METHOD PRIVATE DisposeSelfCreatedNodes : BOOL
VAR
	node : I_Node;
END_VAR
WHILE selfCreatedNodes.TryPop(node) DO
	node.Dispose();
END_WHILE
END_METHOD

METHOD PRIVATE RegisterWithDatatypes
VAR_INPUT
END_VAR
IF datatypes = 0 THEN
	RETURN;
END_IF

datatypes.OnEvent('OnDatatypeAdded', THIS^);
END_METHOD

METHOD PROTECTED CreateAliasArrayBundleNode : I_Node
VAR_INPUT
	NodeDatatype : I_AliasDatatype;
END_VAR
VAR
	pAnyBundleNode : POINTER TO AnyAliasArrayBundleNode;
END_VAR
pAnyBundleNode := __NEW(AnyAliasArrayBundleNode(AliasDatatype := NodeDatatype));
CreateAliasArrayBundleNode := pAnyBundleNode^;
END_METHOD

METHOD PROTECTED CreateAliasArrayUnbundleNode : I_Node
VAR_INPUT
	NodeDatatype : I_AliasDatatype;
END_VAR
VAR
	pAnyUnbundleNode : POINTER TO AnyAliasArrayUnbundleNode;
END_VAR
pAnyUnbundleNode := __NEW(AnyAliasArrayUnbundleNode(AliasDatatype := NodeDatatype));
CreateAliasArrayUnbundleNode := pAnyUnbundleNode^;
END_METHOD

METHOD PROTECTED CreateAliasStructureBundleNode : I_Node
VAR_INPUT
	NodeDatatype : I_AliasDatatype;
END_VAR
VAR
	pAnyBundleNode : POINTER TO AnyAliasStructureBundleNode;
END_VAR
pAnyBundleNode := __NEW(AnyAliasStructureBundleNode(AliasDatatype := NodeDatatype));
CreateAliasStructureBundleNode := pAnyBundleNode^;
END_METHOD

METHOD PROTECTED CreateAliasStructureUnbundleNode : I_Node
VAR_INPUT
	NodeDatatype : I_AliasDatatype;
END_VAR
VAR
	pAnyUnbundleNode : POINTER TO AnyAliasStructureUnbundleNode;
END_VAR
pAnyUnbundleNode := __NEW(AnyAliasStructureUnbundleNode(AliasDatatype := NodeDatatype));
CreateAliasStructureUnbundleNode := pAnyUnbundleNode^;
END_METHOD

METHOD PROTECTED CreateArrayBundleNode : I_Node
VAR_INPUT
	NodeDatatype : I_ArrayDatatype;
END_VAR
VAR
	pAnyBundleNode : POINTER TO AnyArrayBundleNode;
END_VAR
pAnyBundleNode := __NEW(AnyArrayBundleNode(ArrayDatatype := NodeDatatype));
CreateArrayBundleNode := pAnyBundleNode^;
END_METHOD

METHOD PROTECTED CreateArrayUnbundleNode : I_Node
VAR_INPUT
	NodeDatatype : I_ArrayDatatype;
END_VAR
VAR
	pAnyUnbundleNode : POINTER TO AnyArrayUnbundleNode;
END_VAR
pAnyUnbundleNode := __NEW(AnyArrayUnbundleNode(ArrayDatatype := NodeDatatype));
CreateArrayUnbundleNode := pAnyUnbundleNode^;
END_METHOD

METHOD PROTECTED CreateDisplayNode : I_Node
VAR_INPUT
	NodeDatatype : I_Datatype;
END_VAR
VAR
	pAnyDisplayNode : POINTER TO AnyDisplayNode;
END_VAR
pAnyDisplayNode := __NEW(AnyDisplayNode(Datatype := NodeDatatype));
CreateDisplayNode := pAnyDisplayNode^;
END_METHOD

METHOD PROTECTED CreateInterfaceDisplayNode : I_Node
VAR_INPUT
	NodeDatatype : I_InterfaceDatatype;
END_VAR
VAR
	pAnyInterfaceDisplayNode : POINTER TO AnyInterfaceDisplayNode;
END_VAR
pAnyInterfaceDisplayNode := __NEW(AnyInterfaceDisplayNode(Datatype := NodeDatatype));
CreateInterfaceDisplayNode := pAnyInterfaceDisplayNode^;
END_METHOD

METHOD PROTECTED CreateLiteralNode : I_Node
VAR_INPUT
	NodeDatatype : I_Datatype;
END_VAR
VAR
	pAnyLiteralNode : POINTER TO AnyLiteralNode;
END_VAR
pAnyLiteralNode := __NEW(AnyLiteralNode(Datatype := NodeDatatype));
CreateLiteralNode := pAnyLiteralNode^;
END_METHOD

METHOD PROTECTED CreateStructureBundleNode : I_Node
VAR_INPUT
	NodeDatatype : I_StructuredDatatype;
END_VAR
VAR
	pAnyBundleNode : POINTER TO AnyStructureBundleNode;
END_VAR
pAnyBundleNode := __NEW(AnyStructureBundleNode(StructuredDatatype := NodeDatatype));
CreateStructureBundleNode := pAnyBundleNode^;
END_METHOD

METHOD PROTECTED CreateStructureUnbundleNode : I_Node
VAR_INPUT
	NodeDatatype : I_StructuredDatatype;
END_VAR
VAR
	pAnyUnbundleNode : POINTER TO AnyStructureUnbundleNode;
END_VAR
pAnyUnbundleNode := __NEW(AnyStructureUnbundleNode(StructuredDatatype := NodeDatatype));
CreateStructureUnbundleNode := pAnyUnbundleNode^;
END_METHOD

METHOD PROTECTED RegisterAliasArrayBundleNodeOfType
VAR_INPUT
	AliasDatatype : I_AliasDatatype;
END_VAR
VAR
	node : I_Node;
	path : T_MAXSTRING;
END_VAR
node := CreateAliasArrayBundleNode(AliasDatatype);
selfCreatedNodes.Push(node);
path := concat('Bundle/', AliasDatatype.Identifier);
nodeFactory.AddNodeAsPrototype(path,node);
END_METHOD

METHOD PROTECTED RegisterAliasArrayUnbundleNodeOfType
VAR_INPUT
	AliasDatatype : I_AliasDatatype;
END_VAR
VAR
	node : I_Node;
	path : T_MAXSTRING;
END_VAR
node := CreateAliasArrayUnbundleNode(AliasDatatype);
selfCreatedNodes.Push(node);
path := concat('Unbundle/', AliasDatatype.Identifier);
nodeFactory.AddNodeAsPrototype(path,node);
END_METHOD

METHOD PROTECTED RegisterAliasStructureBundleNodeOfType
VAR_INPUT
	AliasDatatype : I_AliasDatatype;
END_VAR
VAR
	node : I_Node;
	path : T_MAXSTRING;
END_VAR
node := CreateAliasStructureBundleNode(AliasDatatype);
selfCreatedNodes.Push(node);
path := concat('Bundle/', AliasDatatype.Identifier);
nodeFactory.AddNodeAsPrototype(path,node);
END_METHOD

METHOD PROTECTED RegisterAliasStructureUnbundleNodeOfType
VAR_INPUT
	AliasDatatype : I_AliasDatatype;
END_VAR
VAR
	node : I_Node;
	path : T_MAXSTRING;
END_VAR
node := CreateAliasStructureUnbundleNode(AliasDatatype);
selfCreatedNodes.Push(node);
path := concat('Unbundle/', AliasDatatype.Identifier);
nodeFactory.AddNodeAsPrototype(path,node);
END_METHOD

METHOD PROTECTED RegisterArrayBundleNodeOfType
VAR_INPUT
	NodeDatatype : I_ArrayDatatype;
END_VAR
VAR
	node : I_Node;
	path : T_MAXSTRING;
END_VAR
node := CreateArrayBundleNode(NodeDatatype);
selfCreatedNodes.Push(node);
path := concat('Bundle/', NodeDatatype.Identifier);
nodeFactory.AddNodeAsPrototype(path,node);
END_METHOD

METHOD PROTECTED RegisterArrayUnbundleNodeOfType
VAR_INPUT
	NodeDatatype : I_ArrayDatatype;
END_VAR
VAR
	node : I_Node;
	path : T_MAXSTRING;
END_VAR
node := CreateArrayUnbundleNode(NodeDatatype);
selfCreatedNodes.Push(node);
path := concat('Unbundle/', NodeDatatype.Identifier);
nodeFactory.AddNodeAsPrototype(path,node);
END_METHOD

METHOD PROTECTED RegisterInterfaceDisplayNodeOfType
VAR_INPUT
	NodeDatatype : I_InterfaceDatatype;
END_VAR
VAR
	node : I_Node;
	path : T_MAXSTRING;
END_VAR
node := CreateInterfaceDisplayNode(NodeDatatype);
selfCreatedNodes.Push(node);
path := concat('Display/', NodeDatatype.Identifier);
nodeFactory.AddNodeAsPrototype(path,node);
END_METHOD

METHOD PROTECTED RegisterInterfaceLiteralNodeOfType
VAR_INPUT
	NodeDatatype : I_InterfaceDatatype;
END_VAR
VAR
	node : I_Node;
	path : T_MAXSTRING;
END_VAR
node := CreateLiteralNode(NodeDatatype);
selfCreatedNodes.Push(node);
path := concat('Literal/', NodeDatatype.Identifier);
nodeFactory.AddNodeAsPrototype(path,node);
END_METHOD

METHOD PROTECTED RegisterPrimitiveDisplayNodeOfType
VAR_INPUT
	NodeDatatype : I_Datatype;
END_VAR
VAR
	node : I_Node;
	path : T_MAXSTRING;
END_VAR
node := CreateDisplayNode(NodeDatatype);
selfCreatedNodes.Push(node);
path := concat('Display/', NodeDatatype.TypeName);
nodeFactory.AddNodeAsPrototype(path,node);
END_METHOD

METHOD PROTECTED RegisterPrimitiveLiteralNodeOfType
VAR_INPUT
	NodeDatatype : I_Datatype;
END_VAR
VAR
	node : I_Node;
	path : T_MAXSTRING;
END_VAR
node := CreateLiteralNode(NodeDatatype);
selfCreatedNodes.Push(node);
path := concat('Literal/', NodeDatatype.TypeName);
nodeFactory.AddNodeAsPrototype(path,node);
END_METHOD

METHOD PROTECTED RegisterStructureBundleNodeOfType
VAR_INPUT
	NodeDatatype : I_StructuredDatatype;
END_VAR
VAR
	node : I_Node;
	path : T_MAXSTRING;
END_VAR
node := CreateStructureBundleNode(NodeDatatype);
selfCreatedNodes.Push(node);
path := concat('Bundle/', NodeDatatype.Identifier);
nodeFactory.AddNodeAsPrototype(path,node);
END_METHOD

METHOD PROTECTED RegisterStructureUnbundleNodeOfType
VAR_INPUT
	NodeDatatype : I_StructuredDatatype;
END_VAR
VAR
	node : I_Node;
	path : T_MAXSTRING;
END_VAR
node := CreateStructureUnbundleNode(NodeDatatype);
selfCreatedNodes.Push(node);
path := concat('Unbundle/', NodeDatatype.Identifier);
nodeFactory.AddNodeAsPrototype(path,node);
END_METHOD

METHOD PROTECTED RegisterUdtDisplayNodeOfType
VAR_INPUT
	NodeDatatype : I_UserDefinedDatatype;
END_VAR
VAR
	node : I_Node;
	path : T_MAXSTRING;
END_VAR
node := CreateDisplayNode(NodeDatatype);
selfCreatedNodes.Push(node);
path := concat('Display/', NodeDatatype.Identifier);
nodeFactory.AddNodeAsPrototype(path,node);
END_METHOD

METHOD PROTECTED RegisterUdtLiteralNodeOfType
VAR_INPUT
	NodeDatatype : I_UserDefinedDatatype;
END_VAR
VAR
	node : I_Node;
	path : T_MAXSTRING;
END_VAR
node := CreateLiteralNode(NodeDatatype);
selfCreatedNodes.Push(node);
path := concat('Literal/', NodeDatatype.Identifier);
nodeFactory.AddNodeAsPrototype(path,node);
END_METHOD

METHOD PUBLIC HandleEvent
VAR_INPUT
	Event : I_Event;
END_VAR
VAR
	datatypeAddedEvent : I_DatatypeAddedEvent;
	primitiveDatatype : I_Datatype;
	aliasDatatypeAddedEvent : I_AliasDatatypeAddedEvent;
	aliasDatatype : I_AliasDatatype;
	enumDatatypeAddedEvent : I_EnumDatatypeAddedEvent;
	enumDatatype : I_EnumDatatype;
	structuredDatatypeAddedEvent : I_StructuredDatatypeAddedEvent;
	structureDatatype : I_StructuredDatatype;
	interfaceDatatypeAddedEvent : I_InterfaceDatatypeAddedEvent;
	interfaceDatatype : I_InterfaceDatatype;
	arrayDatatypeAddedEvent : I_ArrayDatatypeAddedEvent;
	arrayDatatype : I_ArrayDatatype;
END_VAR
IF __QUERYINTERFACE(event, aliasDatatypeAddedEvent) THEN
	aliasDatatype := aliasDatatypeAddedEvent.Target;
	RegisterUdtLiteralNodeOfType(aliasDatatype);
	RegisterUdtDisplayNodeOfType(aliasDatatype);
	
	// at this point we have the lowest level alias who's base type is not alias (or we reached a breakout)
	IF aliasDatatype.Root.TryResolveAsArrayDatatype(arrayDatatype) THEN
		RegisterAliasArrayBundleNodeOfType(aliasDatatype);
		RegisterAliasArrayUnbundleNodeOfType(aliasDatatype);
	ELSIF aliasDatatype.Root.TryResolveAsStructuredDatatype(structureDatatype) THEN
		RegisterAliasStructureBundleNodeOfType(aliasDatatype);
		RegisterAliasStructureUnbundleNodeOfType(aliasDatatype);
	END_IF
		
	RETURN;
END_IF

IF __QUERYINTERFACE(event, enumDatatypeAddedEvent) THEN
	enumDatatype := enumDatatypeAddedEvent.Target;
	RegisterUdtLiteralNodeOfType(enumDatatype);
	RegisterUdtDisplayNodeOfType(enumDatatype);
	RETURN;
END_IF

IF __QUERYINTERFACE(event, interfaceDatatypeAddedEvent) THEN
	interfaceDatatype := interfaceDatatypeAddedEvent.Target;
	RegisterInterfaceLiteralNodeOfType(interfaceDatatype);
	RegisterInterfaceDisplayNodeOfType(interfaceDatatype);
	RETURN;
END_IF

IF __QUERYINTERFACE(event, structuredDatatypeAddedEvent) THEN
	structureDatatype := structuredDatatypeAddedEvent.Target;
	RegisterUdtLiteralNodeOfType(structureDatatype);
	RegisterUdtDisplayNodeOfType(structureDatatype);
	RegisterStructureBundleNodeOfType(structureDatatype);
	RegisterStructureUnbundleNodeOfType(structureDatatype);
	RETURN;
END_IF

IF __QUERYINTERFACE(event, arrayDatatypeAddedEvent) THEN
	RegisterUdtLiteralNodeOfType(arrayDatatypeAddedEvent.Target);
	RegisterUdtDisplayNodeOfType(arrayDatatypeAddedEvent.Target);
	RegisterArrayBundleNodeOfType(arrayDatatypeAddedEvent.Target);
	RegisterArrayUnbundleNodeOfType(arrayDatatypeAddedEvent.Target);
	RETURN;
END_IF

IF __QUERYINTERFACE(event, datatypeAddedEvent) THEN
	primitiveDatatype := datatypeAddedEvent.Target;
	RegisterPrimitiveLiteralNodeOfType(primitiveDatatype);
	RegisterPrimitiveDisplayNodeOfType(primitiveDatatype);
	RETURN;
END_IF
END_METHOD

END_FUNCTION_BLOCK

// Node/Bundle/AnyAliasArrayBundleNode
{attribute 'linkalways'} 
{attribute 'no_explicit_call' := 'This FB is a CLASS and must be accessed using methods or properties'}
{attribute 'enable_dynamic_creation'}
FUNCTION_BLOCK FINAL AnyAliasArrayBundleNode EXTENDS Node
VAR
	in : I_AliasDatatype;
	out : I_AliasDatatype;
	datatypeOperations : DatatypeOperations;
	selfMadeElements : Stack;
END_VAR

METHOD FB_init : BOOL
VAR_INPUT
	bInitRetains : BOOL; // if TRUE, the retain variables are initialized (warm start / cold start)
	bInCopyCode : BOOL;  // if TRUE, the instance afterwards gets moved into the copy code (online change)
	AliasDatatype : I_AliasDatatype;
END_VAR
VAR
	inAsArray : I_ArrayDatatype;
	inAs1D : I_ArrayDatatype_1D;
	inAs2D : I_ArrayDatatype_2D;
	inAs3D : I_ArrayDatatype_3D;
END_VAR
AliasDatatype.Clone().TryResolveAsAliasDatatype(out);
AddOutput('out', out);

AliasDatatype.Clone().TryResolveAsAliasDatatype(in);
in.Root.TryResolveAsArrayDatatype(inAsArray);

IF inAsArray.TryResolveAs1DArrayDatatype(inAs1D) THEN
	ConfigureFor1DArray(inAs1D);
ELSIF inAsArray.TryResolveAs2DArrayDatatype(inAs2D) THEN
	ConfigureFor2DArray(inAs2D);
ELSIF inAsArray.TryResolveAs3DArrayDatatype(inAs3D) THEN
	ConfigureFor3DArray(inAs3D);
END_IF
END_METHOD

METHOD FB_exit : BOOL
VAR_INPUT
	bInCopyCode : BOOL; // if TRUE, the exit method is called for exiting an instance that is copied afterwards (online change).
END_VAR
VAR
	element : I_Datatype;
END_VAR
IF bInCopyCode THEN
	RETURN;
END_IF

in.Dispose();
out.Dispose();
datatypeOperations.Clear();

WHILE selfMadeElements.TryPop(element) DO
	IF element <> 0 THEN 
		element.Dispose();
	END_IF
END_WHILE
END_METHOD

METHOD PRIVATE ConfigureFor1DArray
VAR_INPUT
	array1D : I_ArrayDatatype_1D;
END_VAR
VAR
	lowerBound : DINT;
	upperBound : DINT;
	i : DINT;
	element : I_Datatype;
	elementClone : I_Datatype;
END_VAR
IF NOT array1D.TryGetLowerBound(1, lowerBound) THEN
	RETURN;
END_IF

IF NOT array1D.TryGetUpperBound(1, upperBound) THEN
	RETURN;
END_IF

FOR i := lowerBound TO upperBound DO
	
	IF array1D.TryGetElementAsDatatypeByIndex(i, element) THEN
		elementClone := element.Clone();
		datatypeOperations.AddMemoryCopyOperation(elementClone, element);
		AddParameter(Get1DIndexName(i), elementClone);
		selfMadeElements.Push(elementClone);
	END_IF
	
END_FOR
END_METHOD

METHOD PRIVATE ConfigureFor2DArray
VAR_INPUT
	array2D : I_ArrayDatatype_2D;
END_VAR
VAR
	lowerBoundD1 : DINT;
	upperBoundD1 : DINT;
	lowerBoundD2 : DINT;
	upperBoundD2 : DINT;
	i, j : DINT;
	element : I_Datatype;
	elementClone : I_Datatype;
END_VAR
IF NOT array2D.TryGetLowerBound(1, lowerBoundD1) THEN
	RETURN;
END_IF

IF NOT array2D.TryGetUpperBound(1, upperBoundD1) THEN
	RETURN;
END_IF

IF NOT array2D.TryGetLowerBound(2, lowerBoundD2) THEN
	RETURN;
END_IF

IF NOT array2D.TryGetUpperBound(2, upperBoundD2) THEN
	RETURN;
END_IF

FOR i := lowerBoundD1 TO upperBoundD1 DO
	FOR j := lowerBoundD2 TO upperBoundD2 DO
	
		IF array2D.TryGetElementAsDatatypeByIndex(i, j, element) THEN
			elementClone := element.Clone();
			datatypeOperations.AddMemoryCopyOperation(elementClone, element);
			AddParameter(Get2DIndexName(i,j), elementClone);
			selfMadeElements.Push(elementClone);
		END_IF
	
	END_FOR
END_FOR
END_METHOD

METHOD PRIVATE ConfigureFor3DArray
VAR_INPUT
	array3D : I_ArrayDatatype_3D;
END_VAR
VAR
	lowerBoundD1 : DINT;
	upperBoundD1 : DINT;
	lowerBoundD2 : DINT;
	upperBoundD2 : DINT;
	lowerBoundD3 : DINT;
	upperBoundD3 : DINT;
	i, j, k : DINT;
	element : I_Datatype;
	elementClone : I_Datatype;
END_VAR
IF NOT array3D.TryGetLowerBound(1, lowerBoundD1) THEN
	RETURN;
END_IF

IF NOT array3D.TryGetUpperBound(1, upperBoundD1) THEN
	RETURN;
END_IF

IF NOT array3D.TryGetLowerBound(2, lowerBoundD2) THEN
	RETURN;
END_IF

IF NOT array3D.TryGetUpperBound(2, upperBoundD2) THEN
	RETURN;
END_IF

IF NOT array3D.TryGetLowerBound(3, lowerBoundD3) THEN
	RETURN;
END_IF

IF NOT array3D.TryGetUpperBound(3, upperBoundD3) THEN
	RETURN;
END_IF

FOR i := lowerBoundD1 TO upperBoundD1 DO
	FOR j := lowerBoundD2 TO upperBoundD2 DO
		FOR k := lowerBoundD3 TO upperBoundD3 DO
	
			IF array3D.TryGetElementAsDatatypeByIndex(i, j, k, element) THEN
				elementClone := element.Clone();
				datatypeOperations.AddMemoryCopyOperation(elementClone, element);
				AddParameter(Get3DIndexName(i, j, k), elementClone);
				selfMadeElements.Push(elementClone);
			END_IF
			
		END_FOR
	END_FOR
END_FOR
END_METHOD

METHOD PRIVATE Get1DIndexName : T_MAXSTRING
VAR_INPUT
	Index : DINT;
END_VAR
Get1DIndexName := concat('[', DINT_TO_STRING(Index));
Get1DIndexName := concat(Get1DIndexName, ']');
END_METHOD

METHOD PRIVATE Get2DIndexName : T_MAXSTRING
VAR_INPUT
	Index1 : DINT;
	Index2 : DINT;
END_VAR
Get2DIndexName := concat('[', DINT_TO_STRING(Index1));
Get2DIndexName := concat(Get2DIndexName, ',');
Get2DIndexName := concat(Get2DIndexName, DINT_TO_STRING(Index2));
Get2DIndexName := concat(Get2DIndexName, ']');
END_METHOD

METHOD PRIVATE Get3DIndexName : T_MAXSTRING
VAR_INPUT
	Index1 : DINT;
	Index2 : DINT;
	Index3 : DINT;
END_VAR
Get3DIndexName := concat('[',DINT_TO_STRING(Index1));
Get3DIndexName := concat(Get3DIndexName,',');
Get3DIndexName := concat(Get3DIndexName,DINT_TO_STRING(Index2));
Get3DIndexName := concat(Get3DIndexName,',');
Get3DIndexName := concat(Get3DIndexName,DINT_TO_STRING(Index3));
Get3DIndexName := concat(Get3DIndexName,']');
END_METHOD

METHOD PUBLIC Clone : I_Node
VAR
	pNode : POINTER TO AnyAliasArrayBundleNode;
END_VAR
pNode := __NEW(AnyAliasArrayBundleNode(AliasDatatype := in));
Clone := pNode^;
END_METHOD

METHOD PROTECTED OnExecute
VAR
END_VAR
datatypeOperations.Execute();
memcpy(out.Address, in.Address, in.Size);
END_METHOD

END_FUNCTION_BLOCK

// Node/Unbundle/AnyAliasArrayUnbundleNode
{attribute 'linkalways'} 
{attribute 'no_explicit_call' := 'This FB is a CLASS and must be accessed using methods or properties'}
{attribute 'enable_dynamic_creation'}
FUNCTION_BLOCK FINAL AnyAliasArrayUnbundleNode EXTENDS Node
VAR
	in : I_AliasDatatype;
	out : I_AliasDatatype;
	datatypeOperations : DatatypeOperations;
	selfMadeElements : Stack;
END_VAR

METHOD FB_init : BOOL
VAR_INPUT
	bInitRetains : BOOL; // if TRUE, the retain variables are initialized (warm start / cold start)
	bInCopyCode : BOOL;  // if TRUE, the instance afterwards gets moved into the copy code (online change)
	AliasDatatype : I_AliasDatatype;
END_VAR
VAR
	outAsArray : I_ArrayDatatype;
	outAs1D : I_ArrayDatatype_1D;
	outAs2D : I_ArrayDatatype_2D;
	outAs3D : I_ArrayDatatype_3D;
END_VAR
AliasDatatype.Clone().TryResolveAsAliasDatatype(in);
AddInput('in', in);

AliasDatatype.Clone().TryResolveAsAliasDatatype(out);
out.Root.TryResolveAsArrayDatatype(outAsArray);

IF outAsArray.TryResolveAs1DArrayDatatype(outAs1D) THEN
	ConfigureFor1DArray(outAs1D);
ELSIF outAsArray.TryResolveAs2DArrayDatatype(outAs2D) THEN
	ConfigureFor2DArray(outAs2D);
ELSIF outAsArray.TryResolveAs3DArrayDatatype(outAs3D) THEN
	ConfigureFor3DArray(outAs3D);
END_IF
END_METHOD

METHOD FB_exit : BOOL
VAR_INPUT
	bInCopyCode : BOOL; // if TRUE, the exit method is called for exiting an instance that is copied afterwards (online change).
END_VAR
VAR
	element : I_Datatype;
END_VAR
IF bInCopyCode THEN
	RETURN;
END_IF

in.Dispose();
out.Dispose();
datatypeOperations.Clear();

WHILE selfMadeElements.TryPop(element) DO
	IF element <> 0 THEN 
		element.dispose();
	END_IF
END_WHILE
END_METHOD

METHOD PRIVATE ConfigureFor1DArray
VAR_INPUT
	array1D : I_ArrayDatatype_1D;
END_VAR
VAR
	lowerBound : DINT;
	upperBound : DINT;
	i : DINT;
	element : I_Datatype;
	elementClone : I_Datatype;
END_VAR
IF NOT array1D.TryGetLowerBound(1, lowerBound) THEN
	RETURN;
END_IF

IF NOT array1D.TryGetUpperBound(1, upperBound) THEN
	RETURN;
END_IF

FOR i := lowerBound TO upperBound DO
	
	IF array1D.TryGetElementAsDatatypeByIndex(i, element) THEN
		elementClone := element.Clone();
		datatypeOperations.AddMemoryCopyOperation(element, elementClone);
		AddOutput(Get1DIndexName(i), elementClone);
		selfMadeElements.Push(elementClone);
	END_IF
	
END_FOR
END_METHOD

METHOD PRIVATE ConfigureFor2DArray
VAR_INPUT
	array2D : I_ArrayDatatype_2D;
END_VAR
VAR
	lowerBoundD1 : DINT;
	upperBoundD1 : DINT;
	lowerBoundD2 : DINT;
	upperBoundD2 : DINT;
	i, j : DINT;
	element : I_Datatype;
	elementClone : I_Datatype;
END_VAR
IF NOT array2D.TryGetLowerBound(1, lowerBoundD1) THEN
	RETURN;
END_IF

IF NOT array2D.TryGetUpperBound(1, upperBoundD1) THEN
	RETURN;
END_IF

IF NOT array2D.TryGetLowerBound(2, lowerBoundD2) THEN
	RETURN;
END_IF

IF NOT array2D.TryGetUpperBound(2, upperBoundD2) THEN
	RETURN;
END_IF

FOR i := lowerBoundD1 TO upperBoundD1 DO
	FOR j := lowerBoundD2 TO upperBoundD2 DO
	
		IF array2D.TryGetElementAsDatatypeByIndex(i, j, element) THEN
			elementClone := element.Clone();
			datatypeOperations.AddMemoryCopyOperation(element, elementClone);
			AddOutput(Get2DIndexName(i,j), elementClone);
			selfMadeElements.Push(elementClone);
		END_IF
	
	END_FOR
END_FOR
END_METHOD

METHOD PRIVATE ConfigureFor3DArray
VAR_INPUT
	array3D : I_ArrayDatatype_3D;
END_VAR
VAR
	lowerBoundD1 : DINT;
	upperBoundD1 : DINT;
	lowerBoundD2 : DINT;
	upperBoundD2 : DINT;
	lowerBoundD3 : DINT;
	upperBoundD3 : DINT;
	i, j, k : DINT;
	element : I_Datatype;
	elementClone : I_Datatype;
END_VAR
IF NOT array3D.TryGetLowerBound(1, lowerBoundD1) THEN
	RETURN;
END_IF

IF NOT array3D.TryGetUpperBound(1, upperBoundD1) THEN
	RETURN;
END_IF

IF NOT array3D.TryGetLowerBound(2, lowerBoundD2) THEN
	RETURN;
END_IF

IF NOT array3D.TryGetUpperBound(2, upperBoundD2) THEN
	RETURN;
END_IF

IF NOT array3D.TryGetLowerBound(3, lowerBoundD3) THEN
	RETURN;
END_IF

IF NOT array3D.TryGetUpperBound(3, upperBoundD3) THEN
	RETURN;
END_IF

FOR i := lowerBoundD1 TO upperBoundD1 DO
	FOR j := lowerBoundD2 TO upperBoundD2 DO
		FOR k := lowerBoundD3 TO upperBoundD3 DO
	
			IF array3D.TryGetElementAsDatatypeByIndex(i, j, k, element) THEN
				elementClone := element.Clone();
				datatypeOperations.AddMemoryCopyOperation(element, elementClone);
				AddOutput(Get3DIndexName(i,j,k), elementClone);
				selfMadeElements.Push(elementClone);
			END_IF
			
		END_FOR
	END_FOR
END_FOR
END_METHOD

METHOD PRIVATE Get1DIndexName : T_MAXSTRING
VAR_INPUT
	Index : DINT;
END_VAR
Get1DIndexName := concat('[',DINT_TO_STRING(Index));
Get1DIndexName := concat(Get1DIndexName,']');
END_METHOD

METHOD PRIVATE Get2DIndexName : T_MAXSTRING
VAR_INPUT
	Index1 : DINT;
	Index2 : DINT;
END_VAR
Get2DIndexName := concat('[',DINT_TO_STRING(Index1));
Get2DIndexName := concat(Get2DIndexName,',');
Get2DIndexName := concat(Get2DIndexName,DINT_TO_STRING(Index2));
Get2DIndexName := concat(Get2DIndexName,']');
END_METHOD

METHOD PRIVATE Get3DIndexName : T_MAXSTRING
VAR_INPUT
	Index1 : DINT;
	Index2 : DINT;
	Index3 : DINT;
END_VAR
Get3DIndexName := concat('[',DINT_TO_STRING(Index1));
Get3DIndexName := concat(Get3DIndexName,',');
Get3DIndexName := concat(Get3DIndexName,DINT_TO_STRING(Index2));
Get3DIndexName := concat(Get3DIndexName,',');
Get3DIndexName := concat(Get3DIndexName,DINT_TO_STRING(Index3));
Get3DIndexName := concat(Get3DIndexName,']');
END_METHOD

METHOD PUBLIC Clone : I_Node
VAR
	pNode : POINTER TO AnyAliasArrayUnbundleNode;
END_VAR
pNode := __NEW(AnyAliasArrayUnbundleNode(AliasDatatype := in));
Clone := pNode^;
END_METHOD

METHOD PROTECTED OnExecute
VAR
END_VAR
memcpy(out.Address, in.Address, in.Size);
datatypeOperations.Execute();
END_METHOD

END_FUNCTION_BLOCK

// Node/Bundle/AnyAliasStructureBundleNode
{attribute 'linkalways'} 
{attribute 'no_explicit_call' := 'This FB is a CLASS and must be accessed using methods or properties'}
{attribute 'enable_dynamic_creation'}
FUNCTION_BLOCK FINAL AnyAliasStructureBundleNode EXTENDS Node
VAR
	in : I_AliasDatatype;
	out : I_AliasDatatype;
	datatypeOperations : DatatypeOperations;
	selfMadeMembers : Stack;
END_VAR

METHOD FB_init : BOOL
VAR_INPUT
	bInitRetains : BOOL; // if TRUE, the retain variables are initialized (warm start / cold start)
	bInCopyCode : BOOL;  // if TRUE, the instance afterwards gets moved into the copy code (online change)
	AliasDatatype : I_AliasDatatype;
END_VAR
VAR
	inAsStructured : I_StructuredDatatype;
	enumerator : I_KeyValueForwardEnumerator;
	member : I_Datatype;
	memberAsBit : I_BitDatatype;
	memberAsBool : I_Datatype;
	_bool : pointer to _BOOL;
	memberClone : I_Datatype;
END_VAR
AliasDatatype.Clone().TryResolveAsAliasDatatype(out);
AddOutput('out', out);

AliasDatatype.Clone().TryResolveAsAliasDatatype(in);
in.Root.TryResolveAsStructuredDatatype(inAsStructured);
enumerator := inAsStructured.Members.GetMemberEnumerator();

WHILE enumerator.MoveNext() DO 
	IF enumerator.TryGet(member) THEN
		IF member.TryResolveAsBitDatatype(memberAsBit) THEN
			// if the element is a _bit then this needs to be treated differently (as you cannot simply memcpy
			// a bit, as it sits next to other data. Instead, a bool is added in it's place.	
			_bool := __NEW(_BOOL(InitialValue := memberAsBit.Value));
			datatypeOperations.AddWriteBoolToBitOperation(_bool^, memberAsBit);
			AddParameter(enumerator.Key, _bool^);
			memberAsBool := _bool^;
			selfMadeMembers.Push(memberAsBool);
		ELSE
			// for all other datatypes,
			memberClone := member.Clone();
			datatypeOperations.AddMemoryCopyOperation(memberClone, member);
			AddParameter(enumerator.key, memberClone);
			selfMadeMembers.Push(memberClone);
		END_IF
	END_IF
END_WHILE

enumerator.Dispose();
END_METHOD

METHOD FB_exit : BOOL
VAR_INPUT
	bInCopyCode : BOOL; // if TRUE, the exit method is called for exiting an instance that is copied afterwards (online change).
END_VAR
VAR
	member : I_Datatype;
END_VAR
IF bInCopyCode THEN
	RETURN;
END_IF

in.Dispose();
out.Dispose();
datatypeOperations.Clear();

WHILE selfMadeMembers.TryPop(member) DO
	IF member <> 0 THEN 
		member.dispose();
	END_IF
END_WHILE
END_METHOD

METHOD PUBLIC Clone : I_Node
VAR
	pNode : POINTER TO AnyAliasStructureBundleNode;
END_VAR
pNode := __NEW(AnyAliasStructureBundleNode(AliasDatatype := in));
Clone := pNode^;
END_METHOD

METHOD PROTECTED OnExecute
VAR
END_VAR
datatypeOperations.Execute();
memcpy(out.Address, in.Address, in.Size);
END_METHOD

END_FUNCTION_BLOCK

// Node/Unbundle/AnyAliasStructureUnbundleNode
{attribute 'linkalways'} 
{attribute 'no_explicit_call' := 'This FB is a CLASS and must be accessed using methods or properties'}
{attribute 'enable_dynamic_creation'}
FUNCTION_BLOCK FINAL AnyAliasStructureUnbundleNode EXTENDS Node
VAR
	in : I_AliasDatatype;
	out : I_AliasDatatype;
	datatypeOperations : DatatypeOperations;
	selfMadeMembers : Stack;
END_VAR

METHOD FB_init : BOOL
VAR_INPUT
	bInitRetains : BOOL; // if TRUE, the retain variables are initialized (warm start / cold start)
	bInCopyCode : BOOL;  // if TRUE, the instance afterwards gets moved into the copy code (online change)
	AliasDatatype : I_AliasDatatype;
END_VAR
VAR
	outAsStructure : I_StructuredDatatype;
	enumerator : I_KeyValueForwardEnumerator;
	member : I_Datatype;
	memberAsBit : I_BitDatatype;
	memberAsBool : I_Datatype;
	_bool : Pointer to _BOOL;
	memberClone : I_Datatype;
END_VAR
AliasDatatype.Clone().TryResolveAsAliasDatatype(in);
AddInput('in', in);

AliasDatatype.Clone().TryResolveAsAliasDatatype(out);
out.Root.TryResolveAsStructuredDatatype(outAsStructure);
enumerator := outAsStructure.Members.GetMemberEnumerator();

WHILE enumerator.MoveNext() DO 
	IF enumerator.TryGet(member) THEN
		IF member.TryResolveAsBitDatatype(memberAsBit) THEN
			// if the element is a _bit then this needs to be treated differently (as you cannot simply memcpy
			// a bit, as it sits next to other data. Instead, a bool is added in it's place.	
			_bool := __NEW(_BOOL(InitialValue := memberAsBit.Value));
			datatypeOperations.AddWriteBitToBoolOperation(memberAsBit, _bool^);
			AddOutput(enumerator.Key, _bool^);
			memberAsBool := _bool^;
			selfMadeMembers.Push(memberAsBool);
		ELSE
			// for all other datatypes,
			memberClone := member.Clone();
			datatypeOperations.AddMemoryCopyOperation(member, memberClone);
			AddOutput(enumerator.key, memberClone);
			selfMadeMembers.Push(memberClone);
		END_IF		
	END_IF
END_WHILE

enumerator.Dispose();
END_METHOD

METHOD FB_exit : BOOL
VAR_INPUT
	bInCopyCode : BOOL; // if TRUE, the exit method is called for exiting an instance that is copied afterwards (online change).
END_VAR
VAR
	member : I_Datatype;
END_VAR
IF bInCopyCode THEN
	RETURN;
END_IF

in.Dispose();
out.Dispose();
datatypeOperations.Clear();

WHILE selfMadeMembers.TryPop(member) DO
	IF member <> 0 THEN 
		member.dispose();
	END_IF
END_WHILE
END_METHOD

METHOD PUBLIC Clone : I_Node
VAR
	pNode : POINTER TO AnyAliasStructureUnbundleNode;
END_VAR
pNode := __NEW(AnyAliasStructureUnbundleNode(AliasDatatype := in));
Clone := pNode^;
END_METHOD

METHOD PROTECTED OnExecute
VAR
END_VAR
memcpy(out.Address, in.Address, in.Size);
datatypeOperations.Execute();
END_METHOD

END_FUNCTION_BLOCK

// Node/Bundle/AnyArrayBundleNode
{attribute 'linkalways'} 
{attribute 'no_explicit_call' := 'This FB is a CLASS and must be accessed using methods or properties'}
{attribute 'enable_dynamic_creation'}
FUNCTION_BLOCK FINAL AnyArrayBundleNode EXTENDS Node
VAR
	in : I_ArrayDatatype;
	out : I_ArrayDatatype;
	datatypeOperations : DatatypeOperations;
	selfMadeElements : Stack;
END_VAR

METHOD FB_init : BOOL
VAR_INPUT
	bInitRetains : BOOL; // if TRUE, the retain variables are initialized (warm start / cold start)
	bInCopyCode : BOOL;  // if TRUE, the instance afterwards gets moved into the copy code (online change)
	ArrayDatatype : I_ArrayDatatype;
END_VAR
VAR
	inAs1D : I_ArrayDatatype_1D;
	inAs2D : I_ArrayDatatype_2D;
	inAs3D : I_ArrayDatatype_3D;
END_VAR
ArrayDatatype.Clone().TryResolveAsArrayDatatype(out);
AddOutput('out', out);

ArrayDatatype.Clone().TryResolveAsArrayDatatype(in);

IF in.TryResolveAs1DArrayDatatype(inAs1D) THEN
	ConfigureFor1DArray(inAs1D);
ELSIF in.TryResolveAs2DArrayDatatype(inAs2D) THEN
	ConfigureFor2DArray(inAs2D);
ELSIF in.TryResolveAs3DArrayDatatype(inAs3D) THEN
	ConfigureFor3DArray(inAs3D);
END_IF
END_METHOD

METHOD FB_exit : BOOL
VAR_INPUT
	bInCopyCode : BOOL; // if TRUE, the exit method is called for exiting an instance that is copied afterwards (online change).
END_VAR
VAR
	element : I_Datatype;
END_VAR
IF bInCopyCode THEN
	RETURN;
END_IF

in.Dispose();
out.Dispose();
datatypeOperations.Clear();

WHILE selfMadeElements.TryPop(element) DO
	IF element <> 0 THEN 
		element.dispose();
	END_IF
END_WHILE
END_METHOD

METHOD PRIVATE ConfigureFor1DArray
VAR_INPUT
	array1D : I_ArrayDatatype_1D;
END_VAR
VAR
	lowerBound : DINT;
	upperBound : DINT;
	i : DINT;
	element : I_Datatype;
	elementClone : I_Datatype;
END_VAR
IF NOT array1D.TryGetLowerBound(1, lowerBound) THEN
	RETURN;
END_IF

IF NOT array1D.TryGetUpperBound(1, upperBound) THEN
	RETURN;
END_IF

FOR i := lowerBound TO upperBound DO
	
	IF array1D.TryGetElementAsDatatypeByIndex(i, element) THEN
		elementClone := element.Clone();
		datatypeOperations.AddMemoryCopyOperation(elementClone, element);
		AddParameter(Get1DIndexName(i), elementClone);
		selfMadeElements.Push(elementClone);
	END_IF
	
END_FOR
END_METHOD

METHOD PRIVATE ConfigureFor2DArray
VAR_INPUT
	array2D : I_ArrayDatatype_2D;
END_VAR
VAR
	lowerBoundD1 : DINT;
	upperBoundD1 : DINT;
	lowerBoundD2 : DINT;
	upperBoundD2 : DINT;
	i, j : DINT;
	element : I_Datatype;
	elementClone : I_Datatype;
END_VAR
IF NOT array2D.TryGetLowerBound(1, lowerBoundD1) THEN
	RETURN;
END_IF

IF NOT array2D.TryGetUpperBound(1, upperBoundD1) THEN
	RETURN;
END_IF

IF NOT array2D.TryGetLowerBound(2, lowerBoundD2) THEN
	RETURN;
END_IF

IF NOT array2D.TryGetUpperBound(2, upperBoundD2) THEN
	RETURN;
END_IF

FOR i := lowerBoundD1 TO upperBoundD1 DO
	FOR j := lowerBoundD2 TO upperBoundD2 DO
	
		IF array2D.TryGetElementAsDatatypeByIndex(i, j, element) THEN
			elementClone := element.Clone();
			datatypeOperations.AddMemoryCopyOperation(elementClone, element);
			AddParameter(Get2DIndexName(i,j), elementClone);
			selfMadeElements.Push(elementClone);
		END_IF
	
	END_FOR
END_FOR
END_METHOD

METHOD PRIVATE ConfigureFor3DArray
VAR_INPUT
	array3D : I_ArrayDatatype_3D;
END_VAR
VAR
	lowerBoundD1 : DINT;
	upperBoundD1 : DINT;
	lowerBoundD2 : DINT;
	upperBoundD2 : DINT;
	lowerBoundD3 : DINT;
	upperBoundD3 : DINT;
	i, j, k : DINT;
	element : I_Datatype;
	elementClone : I_Datatype;
END_VAR
IF NOT array3D.TryGetLowerBound(1, lowerBoundD1) THEN
	RETURN;
END_IF

IF NOT array3D.TryGetUpperBound(1, upperBoundD1) THEN
	RETURN;
END_IF

IF NOT array3D.TryGetLowerBound(2, lowerBoundD2) THEN
	RETURN;
END_IF

IF NOT array3D.TryGetUpperBound(2, upperBoundD2) THEN
	RETURN;
END_IF

IF NOT array3D.TryGetLowerBound(3, lowerBoundD3) THEN
	RETURN;
END_IF

IF NOT array3D.TryGetUpperBound(3, upperBoundD3) THEN
	RETURN;
END_IF

FOR i := lowerBoundD1 TO upperBoundD1 DO
	FOR j := lowerBoundD2 TO upperBoundD2 DO
		FOR k := lowerBoundD3 TO upperBoundD3 DO
	
			IF array3D.TryGetElementAsDatatypeByIndex(i, j, k, element) THEN
				elementClone := element.Clone();
				datatypeOperations.AddMemoryCopyOperation(elementClone, element);
				AddParameter(Get3DIndexName(i,j,k), elementClone);
				selfMadeElements.Push(elementClone);
			END_IF
			
		END_FOR
	END_FOR
END_FOR
END_METHOD

METHOD PRIVATE Get1DIndexName : T_MAXSTRING
VAR_INPUT
	Index : DINT;
END_VAR
Get1DIndexName := concat('[',DINT_TO_STRING(Index));
Get1DIndexName := concat(Get1DIndexName,']');
END_METHOD

METHOD PRIVATE Get2DIndexName : T_MAXSTRING
VAR_INPUT
	Index1 : DINT;
	Index2 : DINT;
END_VAR
Get2DIndexName := concat('[',DINT_TO_STRING(Index1));
Get2DIndexName := concat(Get2DIndexName,',');
Get2DIndexName := concat(Get2DIndexName,DINT_TO_STRING(Index2));
Get2DIndexName := concat(Get2DIndexName,']');
END_METHOD

METHOD PRIVATE Get3DIndexName : T_MAXSTRING
VAR_INPUT
	Index1 : DINT;
	Index2 : DINT;
	Index3 : DINT;
END_VAR
Get3DIndexName := concat('[',DINT_TO_STRING(Index1));
Get3DIndexName := concat(Get3DIndexName,',');
Get3DIndexName := concat(Get3DIndexName,DINT_TO_STRING(Index2));
Get3DIndexName := concat(Get3DIndexName,',');
Get3DIndexName := concat(Get3DIndexName,DINT_TO_STRING(Index3));
Get3DIndexName := concat(Get3DIndexName,']');
END_METHOD

METHOD PUBLIC Clone : I_Node
VAR
	pNode : POINTER TO AnyArrayBundleNode;
END_VAR
pNode := __NEW(AnyArrayBundleNode(ArrayDatatype := in));
Clone := pNode^;
END_METHOD

METHOD PROTECTED OnExecute
VAR
END_VAR
datatypeOperations.Execute();
memcpy(out.Address, in.Address, in.Size);
END_METHOD

END_FUNCTION_BLOCK

// Node/Unbundle/AnyArrayUnbundleNode
{attribute 'linkalways'} 
{attribute 'no_explicit_call' := 'This FB is a CLASS and must be accessed using methods or properties'}
{attribute 'enable_dynamic_creation'}
FUNCTION_BLOCK FINAL AnyArrayUnbundleNode EXTENDS Node
VAR
	in : I_ArrayDatatype;
	out : I_ArrayDatatype;
	datatypeOperations : DatatypeOperations;
	selfMadeElements : Stack;
END_VAR

METHOD FB_init : BOOL
VAR_INPUT
	bInitRetains : BOOL; // if TRUE, the retain variables are initialized (warm start / cold start)
	bInCopyCode : BOOL;  // if TRUE, the instance afterwards gets moved into the copy code (online change)
	ArrayDatatype : I_ArrayDatatype;
END_VAR
VAR
	outAs1D : I_ArrayDatatype_1D;
	outAs2D : I_ArrayDatatype_2D;
	outAs3D : I_ArrayDatatype_3D;
END_VAR
ArrayDatatype.Clone().TryResolveAsArrayDatatype(in);
AddInput('in', in);

ArrayDatatype.Clone().TryResolveAsArrayDatatype(out);

IF out.TryResolveAs1DArrayDatatype(outAs1D) THEN
	ConfigureFor1DArray(outAs1D);
ELSIF out.TryResolveAs2DArrayDatatype(outAs2D) THEN
	ConfigureFor2DArray(outAs2D);
ELSIF out.TryResolveAs3DArrayDatatype(outAs3D) THEN
	ConfigureFor3DArray(outAs3D);
END_IF
END_METHOD

METHOD FB_exit : BOOL
VAR_INPUT
	bInCopyCode : BOOL; // if TRUE, the exit method is called for exiting an instance that is copied afterwards (online change).
END_VAR
VAR
	element : I_Datatype;
END_VAR
IF bInCopyCode THEN
	RETURN;
END_IF

in.Dispose();
out.Dispose();
datatypeOperations.Clear();

WHILE selfMadeElements.TryPop(element) DO
	IF element <> 0 THEN 
		element.dispose();
	END_IF
END_WHILE
END_METHOD

METHOD PRIVATE ConfigureFor1DArray
VAR_INPUT
	array1D : I_ArrayDatatype_1D;
END_VAR
VAR
	lowerBound : DINT;
	upperBound : DINT;
	i : DINT;
	element : I_Datatype;
	elementClone : I_Datatype;
END_VAR
IF NOT array1D.TryGetLowerBound(1, lowerBound) THEN
	RETURN;
END_IF

IF NOT array1D.TryGetUpperBound(1, upperBound) THEN
	RETURN;
END_IF

FOR i := lowerBound TO upperBound DO
	
	IF array1D.TryGetElementAsDatatypeByIndex(i, element) THEN
		elementClone := element.Clone();
		datatypeOperations.AddMemoryCopyOperation(element, elementClone);
		AddOutput(Get1DIndexName(i), elementClone);
		selfMadeElements.Push(elementClone);
	END_IF
	
END_FOR
END_METHOD

METHOD PRIVATE ConfigureFor2DArray
VAR_INPUT
	array2D : I_ArrayDatatype_2D;
END_VAR
VAR
	lowerBoundD1 : DINT;
	upperBoundD1 : DINT;
	lowerBoundD2 : DINT;
	upperBoundD2 : DINT;
	i, j : DINT;
	element : I_Datatype;
	elementClone : I_Datatype;
END_VAR
IF NOT array2D.TryGetLowerBound(1, lowerBoundD1) THEN
	RETURN;
END_IF

IF NOT array2D.TryGetUpperBound(1, upperBoundD1) THEN
	RETURN;
END_IF

IF NOT array2D.TryGetLowerBound(2, lowerBoundD2) THEN
	RETURN;
END_IF

IF NOT array2D.TryGetUpperBound(2, upperBoundD2) THEN
	RETURN;
END_IF

FOR i := lowerBoundD1 TO upperBoundD1 DO
	FOR j := lowerBoundD2 TO upperBoundD2 DO
	
		IF array2D.TryGetElementAsDatatypeByIndex(i, j, element) THEN
			elementClone := element.Clone();
			datatypeOperations.AddMemoryCopyOperation(element, elementClone);
			AddOutput(Get2DIndexName(i,j), elementClone);
			selfMadeElements.Push(elementClone);
		END_IF
	
	END_FOR
END_FOR
END_METHOD

METHOD PRIVATE ConfigureFor3DArray
VAR_INPUT
	array3D : I_ArrayDatatype_3D;
END_VAR
VAR
	lowerBoundD1 : DINT;
	upperBoundD1 : DINT;
	lowerBoundD2 : DINT;
	upperBoundD2 : DINT;
	lowerBoundD3 : DINT;
	upperBoundD3 : DINT;
	i, j, k : DINT;
	element : I_Datatype;
	elementClone : I_Datatype;
END_VAR
IF NOT array3D.TryGetLowerBound(1, lowerBoundD1) THEN
	RETURN;
END_IF

IF NOT array3D.TryGetUpperBound(1, upperBoundD1) THEN
	RETURN;
END_IF

IF NOT array3D.TryGetLowerBound(2, lowerBoundD2) THEN
	RETURN;
END_IF

IF NOT array3D.TryGetUpperBound(2, upperBoundD2) THEN
	RETURN;
END_IF

IF NOT array3D.TryGetLowerBound(3, lowerBoundD3) THEN
	RETURN;
END_IF

IF NOT array3D.TryGetUpperBound(3, upperBoundD3) THEN
	RETURN;
END_IF

FOR i := lowerBoundD1 TO upperBoundD1 DO
	FOR j := lowerBoundD2 TO upperBoundD2 DO
		FOR k := lowerBoundD3 TO upperBoundD3 DO
	
			IF array3D.TryGetElementAsDatatypeByIndex(i, j, k, element) THEN
				elementClone := element.Clone();
				datatypeOperations.AddMemoryCopyOperation(element, elementClone);
				AddOutput(Get3DIndexName(i,j,k), elementClone);
				selfMadeElements.Push(elementClone);
			END_IF
			
		END_FOR
	END_FOR
END_FOR
END_METHOD

METHOD PRIVATE Get1DIndexName : T_MAXSTRING
VAR_INPUT
	Index : DINT;
END_VAR
Get1DIndexName := concat('[',DINT_TO_STRING(Index));
Get1DIndexName := concat(Get1DIndexName,']');
END_METHOD

METHOD PRIVATE Get2DIndexName : T_MAXSTRING
VAR_INPUT
	Index1 : DINT;
	Index2 : DINT;
END_VAR
Get2DIndexName := concat('[',DINT_TO_STRING(Index1));
Get2DIndexName := concat(Get2DIndexName,',');
Get2DIndexName := concat(Get2DIndexName,DINT_TO_STRING(Index2));
Get2DIndexName := concat(Get2DIndexName,']');
END_METHOD

METHOD PRIVATE Get3DIndexName : T_MAXSTRING
VAR_INPUT
	Index1 : DINT;
	Index2 : DINT;
	Index3 : DINT;
END_VAR
Get3DIndexName := concat('[',DINT_TO_STRING(Index1));
Get3DIndexName := concat(Get3DIndexName,',');
Get3DIndexName := concat(Get3DIndexName,DINT_TO_STRING(Index2));
Get3DIndexName := concat(Get3DIndexName,',');
Get3DIndexName := concat(Get3DIndexName,DINT_TO_STRING(Index3));
Get3DIndexName := concat(Get3DIndexName,']');
END_METHOD

METHOD PUBLIC Clone : I_Node
VAR
	pNode : POINTER TO AnyArrayUnbundleNode;
END_VAR
pNode := __NEW(AnyArrayUnbundleNode(ArrayDatatype := in));
Clone := pNode^;
END_METHOD

METHOD PROTECTED OnExecute
VAR
END_VAR
memcpy(out.Address, in.Address, in.Size);
datatypeOperations.Execute();
END_METHOD

END_FUNCTION_BLOCK

// Node/Display/AnyDisplayNode
{attribute 'linkalways'} 
{attribute 'no_explicit_call' := 'This FB is a CLASS and must be accessed using methods or properties'}
{attribute 'enable_dynamic_creation'}
FUNCTION_BLOCK FINAL AnyDisplayNode EXTENDS Node
VAR
	in : I_Datatype;
	display : I_Datatype;
END_VAR

METHOD FB_init : BOOL
VAR_INPUT
	bInitRetains : BOOL; // if TRUE, the retain variables are initialized (warm start / cold start)
	bInCopyCode : BOOL;  // if TRUE, the instance afterwards gets moved into the copy code (online change)
	Datatype : I_Datatype;
END_VAR
THIS^.in := Datatype.Clone();
THIS^.display := Datatype.Clone();

AddInput('in', THIS^.in);
AddContent('display', THIS^.display);
END_METHOD

METHOD FB_exit : BOOL
VAR_INPUT
	bInCopyCode : BOOL; // if TRUE, the exit method is called for exiting an instance that is copied afterwards (online change).
END_VAR
IF bInCopyCode THEN
	RETURN;
END_IF

in.Dispose();
display.Dispose();
END_METHOD

METHOD PUBLIC Clone : I_Node
VAR
	pNode : POINTER TO AnyDisplayNode;
END_VAR
pNode := __NEW(AnyDisplayNode(Datatype := in));
Clone := pNode^;
END_METHOD

METHOD PROTECTED OnExecute
VAR
END_VAR
memcpy(display.Address, in.Address, in.Size);
END_METHOD

END_FUNCTION_BLOCK

// Node/Display/AnyInterfaceDisplayNode
{attribute 'linkalways'} 
{attribute 'no_explicit_call' := 'This FB is a CLASS and must be accessed using methods or properties'}
{attribute 'enable_dynamic_creation'}
FUNCTION_BLOCK FINAL AnyInterfaceDisplayNode EXTENDS Node
VAR
	in : I_InterfaceDatatype;
	display : I_InterfaceDatatype;
END_VAR

METHOD FB_init : BOOL
VAR_INPUT
	bInitRetains : BOOL; // if TRUE, the retain variables are initialized (warm start / cold start)
	bInCopyCode : BOOL;  // if TRUE, the instance afterwards gets moved into the copy code (online change)
	Datatype : I_InterfaceDatatype;
END_VAR
Datatype.Clone().TryResolveAsInterfaceDatatype(THIS^.in);
Datatype.Clone().TryResolveAsInterfaceDatatype(THIS^.display);

AddInput('in', THIS^.in);
AddContent('display', THIS^.display);
END_METHOD

METHOD FB_exit : BOOL
VAR_INPUT
	bInCopyCode : BOOL; // if TRUE, the exit method is called for exiting an instance that is copied afterwards (online change).
END_VAR
IF bInCopyCode THEN
	RETURN;
END_IF

in.Dispose();
display.Dispose();
END_METHOD

METHOD PUBLIC Clone : I_Node
VAR
	pNode : POINTER TO AnyInterfaceDisplayNode;
END_VAR
pNode := __NEW(AnyInterfaceDisplayNode(Datatype := in));
Clone := pNode^;
END_METHOD

METHOD PROTECTED OnExecute
VAR
END_VAR
display.TryCopyContentFrom(in);
END_METHOD

END_FUNCTION_BLOCK

// Node/Literal/AnyLiteralNode
{attribute 'linkalways'} 
{attribute 'no_explicit_call' := 'This FB is a CLASS and must be accessed using methods or properties'}
{attribute 'enable_dynamic_creation'}
FUNCTION_BLOCK FINAL AnyLiteralNode EXTENDS Node
VAR
	value : I_Datatype;
	out : I_Datatype;
	
	// meta
	suppressInputPort : _BOOL(TRUE);
END_VAR

METHOD FB_init : BOOL
VAR_INPUT
	bInitRetains : BOOL; // if TRUE, the retain variables are initialized (warm start / cold start)
	bInCopyCode : BOOL;  // if TRUE, the instance afterwards gets moved into the copy code (online change)
	Datatype : I_Datatype;
END_VAR
THIS^.value := Datatype.Clone();
THIS^.out := Datatype.Clone();

AddParameter('value', THIS^.value)
	.AddMetadata('suppressInput', suppressInputPort); // literals should not use input ports if available. 
	
AddOutput('out', THIS^.out);
END_METHOD

METHOD FB_exit : BOOL
VAR_INPUT
	bInCopyCode : BOOL; // if TRUE, the exit method is called for exiting an instance that is copied afterwards (online change).
END_VAR
IF bInCopyCode THEN
	RETURN;
END_IF

value.Dispose();
out.Dispose();
END_METHOD

METHOD PUBLIC Clone : I_Node
VAR
	pNode : POINTER TO AnyLiteralNode;
END_VAR
pNode := __NEW(AnyLiteralNode(Datatype := value));
Clone := pNode^;
END_METHOD

METHOD PROTECTED OnExecute
VAR
END_VAR
memcpy(out.Address, value.Address, value.Size);
END_METHOD

END_FUNCTION_BLOCK

// Node/Bundle/AnyStructureBundleNode
{attribute 'linkalways'} 
{attribute 'no_explicit_call' := 'This FB is a CLASS and must be accessed using methods or properties'}
{attribute 'enable_dynamic_creation'}
FUNCTION_BLOCK FINAL AnyStructureBundleNode EXTENDS Node
VAR
	in : I_StructuredDatatype;
	out : I_StructuredDatatype;
	datatypeOperations : DatatypeOperations;
	selfMadeMembers : Stack;
END_VAR

METHOD FB_init : BOOL
VAR_INPUT
	bInitRetains : BOOL; // if TRUE, the retain variables are initialized (warm start / cold start)
	bInCopyCode : BOOL;  // if TRUE, the instance afterwards gets moved into the copy code (online change)
	StructuredDatatype : I_StructuredDatatype;
END_VAR
VAR
	enumerator : I_KeyValueForwardEnumerator;
	member : I_Datatype;
	memberAsBit : I_BitDatatype;
	memberAsBool : I_Datatype;
	_bool : pointer to _BOOL;
	memberClone : I_Datatype;
END_VAR
StructuredDatatype.Clone().TryResolveAsStructuredDatatype(out);
AddOutput('out', out);

StructuredDatatype.Clone().TryResolveAsStructuredDatatype(in);
enumerator := in.Members.GetMemberEnumerator();

WHILE enumerator.MoveNext() DO 
	IF enumerator.TryGet(member) THEN
		IF member.TryResolveAsBitDatatype(memberAsBit) THEN
			// if the element is a _bit then this needs to be treated differently (as you cannot simply memcpy
			// a bit, as it sits next to other data. Instead, a bool is added in it's place.	
			_bool := __NEW(_BOOL(InitialValue := memberAsBit.Value));
			datatypeOperations.AddWriteBoolToBitOperation(_bool^, memberAsBit);
			AddParameter(enumerator.Key, _bool^);
			memberAsBool := _bool^;
			selfMadeMembers.Push(memberAsBool);
		ELSE
			// for all other datatypes,
			memberClone := member.Clone();
			datatypeOperations.AddMemoryCopyOperation(memberClone, member);
			AddParameter(enumerator.key, memberClone);
			selfMadeMembers.Push(memberClone);
		END_IF
	END_IF
END_WHILE

enumerator.Dispose();
END_METHOD

METHOD FB_exit : BOOL
VAR_INPUT
	bInCopyCode : BOOL; // if TRUE, the exit method is called for exiting an instance that is copied afterwards (online change).
END_VAR
VAR
	member : I_Datatype;
END_VAR
IF bInCopyCode THEN
	RETURN;
END_IF

in.Dispose();
out.Dispose();
datatypeOperations.Clear();

WHILE selfMadeMembers.TryPop(member) DO
	IF member <> 0 THEN 
		member.dispose();
	END_IF
END_WHILE
END_METHOD

METHOD PUBLIC Clone : I_Node
VAR
	pNode : POINTER TO AnyStructureBundleNode;
END_VAR
pNode := __NEW(AnyStructureBundleNode(StructuredDatatype := in));
Clone := pNode^;
END_METHOD

METHOD PROTECTED OnExecute
VAR
END_VAR
datatypeOperations.Execute();
memcpy(out.Address, in.Address, in.Size);
END_METHOD

END_FUNCTION_BLOCK

// Node/Unbundle/AnyStructureUnbundleNode
{attribute 'linkalways'} 
{attribute 'no_explicit_call' := 'This FB is a CLASS and must be accessed using methods or properties'}
{attribute 'enable_dynamic_creation'}
FUNCTION_BLOCK FINAL AnyStructureUnbundleNode EXTENDS Node
VAR
	in : I_StructuredDatatype;
	out : I_StructuredDatatype;
	datatypeOperations : DatatypeOperations;
	selfMadeMembers : Stack;
END_VAR

METHOD FB_init : BOOL
VAR_INPUT
	bInitRetains : BOOL; // if TRUE, the retain variables are initialized (warm start / cold start)
	bInCopyCode : BOOL;  // if TRUE, the instance afterwards gets moved into the copy code (online change)
	StructuredDatatype : I_StructuredDatatype;
END_VAR
VAR
	enumerator : I_KeyValueForwardEnumerator;
	member : I_Datatype;
	memberAsBit : I_BitDatatype;
	memberAsBool : I_Datatype;
	_bool : Pointer to _BOOL;
	memberClone : I_Datatype;
END_VAR
StructuredDatatype.Clone().TryResolveAsStructuredDatatype(in);
AddInput('in', in);

StructuredDatatype.Clone().TryResolveAsStructuredDatatype(out);
enumerator := out.Members.GetMemberEnumerator();

WHILE enumerator.MoveNext() DO 
	IF enumerator.TryGet(member) THEN
		IF member.TryResolveAsBitDatatype(memberAsBit) THEN
			// if the element is a _bit then this needs to be treated differently (as you cannot simply memcpy
			// a bit, as it sits next to other data. Instead, a bool is added in it's place.	
			_bool := __NEW(_BOOL(InitialValue := memberAsBit.Value));
			datatypeOperations.AddWriteBitToBoolOperation(memberAsBit, _bool^);
			AddOutput(enumerator.Key, _bool^);
			memberAsBool := _bool^;
			selfMadeMembers.Push(memberAsBool);
		ELSE
			// for all other datatypes,
			memberClone := member.Clone();
			datatypeOperations.AddMemoryCopyOperation(member, memberClone);
			AddOutput(enumerator.key, memberClone);
			selfMadeMembers.Push(memberClone);
		END_IF		
	END_IF
END_WHILE

enumerator.Dispose();
END_METHOD

METHOD FB_exit : BOOL
VAR_INPUT
	bInCopyCode : BOOL; // if TRUE, the exit method is called for exiting an instance that is copied afterwards (online change).
END_VAR
VAR
	member : I_Datatype;
END_VAR
IF bInCopyCode THEN
	RETURN;
END_IF

in.Dispose();
out.Dispose();
datatypeOperations.Clear();

WHILE selfMadeMembers.TryPop(member) DO
	IF member <> 0 THEN 
		member.dispose();
	END_IF
END_WHILE
END_METHOD

METHOD PUBLIC Clone : I_Node
VAR
	pNode : POINTER TO AnyStructureUnbundleNode;
END_VAR
pNode := __NEW(AnyStructureUnbundleNode(StructuredDatatype := in));
Clone := pNode^;
END_METHOD

METHOD PROTECTED OnExecute
VAR
END_VAR
memcpy(out.Address, in.Address, in.Size);
datatypeOperations.Execute();
END_METHOD

END_FUNCTION_BLOCK

// Graph/Base/Graph
{attribute 'linkalways'} 
{attribute 'no_explicit_call' := 'This FB is a CLASS and must be accessed using methods or properties'}
{attribute 'enable_dynamic_creation'}
FUNCTION_BLOCK Graph EXTENDS Disposable IMPLEMENTS I_Graph
VAR
	nodeFactory : I_NodeFactory;
	_uuid : T_MAXSTRING;	
	eventEmitter : EventEmitter;
	nodeHost : NodeHost(THIS^, eventEmitter);
	inputPortHost : InputPortHost(THIS^, eventEmitter);
	outputPortHost : OutputPortHost(THIS^, eventEmitter);
	parameterHost : ParameterHost(THIS^, eventEmitter);
	contentHost : ContentHost(THIS^, eventEmitter);
	alarmHost : AlarmHost(THIS^, eventEmitter);
	metadataHost : MetadataHost(THIS^, eventEmitter);
	extensionHost : ExtensionHost(THIS^,eventEmitter);
	selfCreatedNodes : Stack;
	nodelinks : NodeLinks;
	
	deserializationFailedAlarm : DeserializationFailedAlarm(THIS^);
	deserializationFailedNodeNotSupportedAlarm : DeserializationFailedNodeNotSupportedAlarm(THIS^);
END_VAR

METHOD FB_init : BOOL
VAR_INPUT
	bInitRetains : BOOL; // if TRUE, the retain variables are initialized (warm start / cold start)
	bInCopyCode : BOOL;  // if TRUE, the instance afterwards gets moved into the copy code (online change)
	NodeFactory : I_NodeFactory;
END_VAR
THIS^.nodeFactory := NodeFactory;
END_METHOD

METHOD FB_exit : BOOL
VAR_INPUT
	bInCopyCode : BOOL; // if TRUE, the exit method is called for exiting an instance that is copied afterwards (online change).
END_VAR
IF bInCopyCode THEN
	RETURN;
END_IF

Reset();
END_METHOD

METHOD PRIVATE DisposeSelfCreatedNodes : BOOL
VAR
	node : I_Node;
END_VAR
WHILE selfCreatedNodes.TryPop(node) DO
	nodeHost.RemoveNode(node);
	node.Dispose();
END_WHILE
END_METHOD

METHOD PRIVATE TryConnectLinksInExecutionOrder : BOOL
VAR_INPUT
END_VAR
VAR
	nodeEnumerator : I_ForwardEnumerator;
	linkEnumerator : I_KeyValueForwardEnumerator;
	nodeId : T_MAXSTRING;
	node : I_Node;
	link : I_NodeLink;
END_VAR
nodeEnumerator := nodes.GetNodesInOrderEnumerator();
linkEnumerator := nodelinks.GetKeyValueEnumerator();

WHILE (nodeEnumerator.MoveNext()) DO
	
	IF nodeEnumerator.TryGet(node) THEN
		nodeId := node.Id;
		linkEnumerator.Reset();
		
		WHILE (linkEnumerator.MoveNext()) DO
	
			IF linkEnumerator.TryGet(link) AND_THEN link.SourceNode.Id = nodeId THEN
				IF NOT link.TryConnect() THEN
					linkEnumerator.Dispose();
					nodeEnumerator.Dispose();
					RETURN;	
				END_IF
			END_IF
		
		END_WHILE

	END_IF

END_WHILE

linkEnumerator.Dispose();
nodeEnumerator.Dispose();
TryConnectLinksInExecutionOrder := TRUE;
END_METHOD

METHOD PUBLIC TryDeserializeNodeLinks : BOOL
VAR_INPUT
	Deserializer : I_Deserializer;
	Feedback : I_DeserializerFeedback;
END_VAR
VAR
	linksDeserializer : I_Deserializer;
	linksEnumerator : I_DeserializerArrayForwardEnumerator;
	linkDeserializer : I_Deserializer;
	linkId : T_MAXSTRING;
	sourceNodeId : T_MAXSTRING;
	sourceName : T_MAXSTRING;
	destinationNodeId : T_MAXSTRING;
	destinationName : T_MAXSTRING;
	sourceNode : I_Node;
	sourcePort : I_OutputPort;
	destinationNode : I_Node;
	destinationPort : I_InputPort;
	destinationParameter : I_Parameter;
	link : I_NodeLink;
END_VAR
linksDeserializer := Deserializer.GetKeyArray('links');
linksEnumerator := linksDeserializer.GetArrayEnumerator();

WHILE linksEnumerator.MoveNext() DO
	
	linkDeserializer := linksEnumerator.Current.GetArray();
	
	IF NOT linkDeserializer.GetElementByIndex(0).TryGetString(linkId, Feedback) THEN
		DeserializationFailedAlarm.Raise('Missing linkid from link');
		linksEnumerator.Dispose();
		RETURN;
	END_IF
	
	IF NOT linkDeserializer.GetElementByIndex(1).TryGetString(sourceNodeId, Feedback) THEN
		DeserializationFailedAlarm.Raise('Missing source node id from link');
		linksEnumerator.Dispose();
		RETURN;
	END_IF
	
	IF NOT linkDeserializer.GetElementByIndex(2).TryGetString(sourceName, Feedback) THEN
		DeserializationFailedAlarm.Raise('Missing source name from link');
		linksEnumerator.Dispose();
		RETURN;
	END_IF
	
	IF NOT linkDeserializer.GetElementByIndex(3).TryGetString(destinationNodeId, Feedback) THEN
		DeserializationFailedAlarm.Raise('Missing destination node id from link');
		linksEnumerator.Dispose();
		RETURN;
	END_IF
	
	IF NOT linkDeserializer.GetElementByIndex(4).TryGetString(destinationName, Feedback) THEN
		DeserializationFailedAlarm.Raise('Missing destination name from link');
		linksEnumerator.Dispose();
		RETURN;
	END_IF
	
	IF NOT nodeHost.TryGetNodeById(sourceNodeId, sourceNode) THEN
		DeserializationFailedAlarm.Raise('Unable to get source node when creating link');
		linksEnumerator.Dispose();
		RETURN;
	END_IF
	
	IF NOT nodeHost.TryGetNodeById(destinationNodeId, destinationNode) THEN
		DeserializationFailedAlarm.Raise('Unable to get destination node when creating link');
		linksEnumerator.Dispose();
		RETURN;
	END_IF
	
	IF NOT sourceNode.OutputPorts.TryGetOutputPortByName(sourceName, sourcePort) THEN
		DeserializationFailedAlarm.Raise('Unable to get source when creating link');
		linksEnumerator.Dispose();
		RETURN;
	END_IF
	
	// first try to find the name in the node input ports, then by node parameters
	IF destinationNode.InputPorts.TryGetInputPortByName(destinationName, destinationPort) THEN
		nodelinks.Create(linkId, sourceNode, sourcePort, destinationNode, destinationPort);
	ELSIF  destinationNode.Parameters.TryGetParameterByName(destinationName, destinationParameter) THEN
		nodelinks.Create(linkId, sourceNode, sourcePort, destinationNode, destinationParameter);
	ELSE
		DeserializationFailedAlarm.Raise('Unable to get destination port when creating link');
		linksEnumerator.Dispose();
		RETURN;
	END_IF
	

END_WHILE

IF NOT TryConnectLinksInExecutionOrder() THEN
	DeserializationFailedAlarm.Raise('Unable to finalise links');
	linksEnumerator.Dispose();
	RETURN;
END_IF

TryDeserializeNodeLinks := TRUE;
linksEnumerator.Dispose();
END_METHOD

METHOD PUBLIC TryDeserializeNodes : BOOL;
VAR_INPUT
	Deserializer : I_Deserializer;
	Feedback : I_DeserializerFeedback;
END_VAR
VAR
	nodeDeserializer : I_Deserializer;
	nodesEnumerator : I_DeserializerArrayForwardEnumerator;
	nodeType : T_MAXSTRING;
	pError : POINTER TO MissingNodePrototypeDeserializationError;
	node : I_Node;
END_VAR
nodeDeserializer := Deserializer.GetKeyArray('nodes');
nodesEnumerator := nodeDeserializer.GetArrayEnumerator();

WHILE nodesEnumerator.MoveNext() DO
	
	IF NOT nodesEnumerator.Current.TryGetKeyString('type',nodeType, Feedback) THEN
		RETURN;
	END_IF
	
	IF NOT nodeFactory.TryCreateNodeByType(nodeType, node) THEN
		pError := __NEW(MissingNodePrototypeDeserializationError(MissingType := nodeType));
		Feedback.LogError(pError^);
		DeserializationFailedNodeNotSupportedAlarm.Raise(nodeType);
		nodesEnumerator.Dispose();
		RETURN;
	END_IF
	
	selfCreatedNodes.Push(node);
	
	IF NOT node.TryDeserializeFrom(nodesEnumerator.Current, Feedback) THEN
		DeserializationFailedAlarm.Raise('Node failed to deserialize');
		nodesEnumerator.Dispose();
		RETURN;
	END_IF
	
	Nodes.AddNode(node);

END_WHILE

TryDeserializeNodes := TRUE;
nodesEnumerator.Dispose();
END_METHOD

METHOD PUBLIC Accept
VAR_INPUT
	Visitor : I_GraphVisitor;
END_VAR
Visitor.VisitGraph(THIS^);
END_METHOD

METHOD PUBLIC AddMetadata : I_HostMetadata
VAR_INPUT
	Name : T_MAXSTRING;
	Data : I_Datatype;
END_VAR
Metadatum.AddDataAsMetadata(Name, Data);
AddMetadata := THIS^;
END_METHOD

PROPERTY PUBLIC Alarms : I_Alarms
GET
Alarms := alarmHost;
END_GET
END_PROPERTY

PROPERTY PUBLIC Contents : I_Contents
GET
Contents := contentHost;
END_GET
END_PROPERTY

METHOD Execute
VAR_INPUT
END_VAR
nodeHost.Execute();
END_METHOD

PROPERTY PUBLIC Extensions : I_Extensions
GET
Extensions := extensionHost;
END_GET
END_PROPERTY

PROPERTY PUBLIC HasRaisedAlarm : BOOL
GET
HasRaisedAlarm := alarmHost.HasRaisedAlarm;
END_GET
END_PROPERTY

PROPERTY PUBLIC InputPorts : I_InputPorts
GET
InputPorts := inputPortHost;
END_GET
END_PROPERTY

PROPERTY PUBLIC Metadatum : I_Metadatum
GET
Metadatum := metadataHost;
END_GET
END_PROPERTY

PROPERTY PUBLIC Nodes : I_Nodes
GET
Nodes := nodeHost;
END_GET
END_PROPERTY

METHOD PUBLIC OffEvent
VAR_INPUT
	EventName : T_MaxString;
	EventHandler : I_EventHandler;
END_VAR
eventEmitter.OffEvent(EventName, EventHandler);
END_METHOD

METHOD PUBLIC OnceEvent
VAR_INPUT
	EventName : T_MaxString;
	EventHandler : I_EventHandler;
END_VAR
eventEmitter.OnceEvent(EventName, EventHandler);
END_METHOD

METHOD PUBLIC OnEvent
VAR_INPUT
	EventName : T_MaxString;
	EventHandler : I_EventHandler;
END_VAR
eventEmitter.OnEvent(EventName, EventHandler);
END_METHOD

PROPERTY PUBLIC OutputPorts : I_OutputPorts
GET
OutputPorts := outputPortHost;
END_GET
END_PROPERTY

PROPERTY PUBLIC Parameters : I_Parameters
GET
Parameters := parameterHost;
END_GET
END_PROPERTY

METHOD PUBLIC Reset
VAR_INPUT
END_VAR
_uuid := '';
nodeLinks.Clear();
DisposeSelfCreatedNodes();
END_METHOD

METHOD PUBLIC SerializeWith
VAR_INPUT
	Serializer : I_Serializer;
END_VAR
Serializer.StartObject();
Serializer.AddKeyString('uuid',_uuid);
inputPortHost.SerializeWith(Serializer);
outputPortHost.SerializeWith(Serializer);
parameterHost.SerializeWith(Serializer);
contentHost.SerializeWith(Serializer);
alarmHost.SerializeWith(Serializer);
extensionHost.SerializeWith(Serializer);
metadataHost.SerializeWith(Serializer);
nodeHost.SerializeWith(Serializer);
Serializer.EndObject();
END_METHOD

METHOD PUBLIC TryDeserializeFrom : BOOL
VAR_INPUT
	Deserializer : I_Deserializer;
	Feedback : I_DeserializerFeedback;
END_VAR
VAR
	receivedUuid : T_MAXSTRING;
END_VAR
DeserializationFailedNodeNotSupportedAlarm.Clear();
DeserializationFailedAlarm.Clear();

IF NOT parameterHost.TryDeserializeFrom(Deserializer, Feedback) THEN
	RETURN;
END_IF

IF NOT extensionHost.TryDeserializeFrom(Deserializer, Feedback) THEN
	RETURN;
END_IF

IF NOT Deserializer.TryGetKeyString('uuid', receivedUuid, Feedback) THEN
	RETURN;
END_IF

Reset();

IF NOT TryDeserializeNodes(Deserializer, Feedback) THEN 
	RETURN;
END_IF

IF NOT TryDeserializeNodeLinks(Deserializer, Feedback) THEN
	RETURN;
END_IF

_uuid := receivedUuid;
TryDeserializeFrom := TRUE;
END_METHOD

PROPERTY PUBLIC Uuid : T_MAXSTRING
GET
Uuid := _uuid;
END_GET
END_PROPERTY

END_FUNCTION_BLOCK

// Node/Host/NodeHost
{attribute 'linkalways'} 
{attribute 'no_explicit_call' := 'This FB is a CLASS and must be accessed using methods or properties'}
{attribute 'enable_dynamic_creation'}
FUNCTION_BLOCK NodeHost IMPLEMENTS I_Nodes, I_Serializable
VAR
	hostParent : I_HostNodes;
	eventTarget : I_EventTarget;
	nodes : OrderedDictionary;
	nodesInExecutionOrder : LinkedList;
	executeEnumerator : I_ForwardEnumerator;
END_VAR

METHOD FB_init : BOOL
VAR_INPUT
	bInitRetains : BOOL; // if TRUE, the retain variables are initialized (warm start / cold start)
	bInCopyCode : BOOL;  // if TRUE, the instance afterwards gets moved into the copy code (online change)
	Parent : I_HostNodes;
	parentEventTarget : I_EventTarget;
END_VAR
hostParent := Parent;
eventTarget := parentEventTarget;
CreateExecuteEnumerator();
END_METHOD

METHOD FB_exit : BOOL
VAR_INPUT
	bInCopyCode : BOOL; // if TRUE, the exit method is called for exiting an instance that is copied afterwards (online change).
END_VAR
IF bInCopyCode THEN
	RETURN;
END_IF

DestroyExecuteEnumerator();
END_METHOD

METHOD PRIVATE CreateExecuteEnumerator
VAR_INPUT
END_VAR
IF executeEnumerator <> 0 THEN
	executeEnumerator.Dispose();
END_IF

executeEnumerator := nodesInExecutionOrder.GetEnumerator();
END_METHOD

METHOD PRIVATE DestroyExecuteEnumerator
VAR_INPUT
END_VAR
IF executeEnumerator <> 0 THEN
	executeEnumerator.Dispose();
END_IF
END_METHOD

METHOD PROTECTED EmitOnNodeAddedEvent
VAR_INPUT
	Node : I_Node;
END_VAR
VAR
	nodeAddedEvent : NodeAddedEvent(Target := Node);
END_VAR
IF eventTarget = 0 THEN
	RETURN;
END_IF

eventTarget.Emit('OnNodeAdded', nodeAddedEvent);
END_METHOD

METHOD PROTECTED UpdateExecutionOrder
VAR_INPUT
	Node : I_Node;
END_VAR
VAR
	currentPosition : I_LinkedListNode;
	currentNode : I_Node;
END_VAR
// is the list empty?
IF nodesInExecutionOrder.First = 0 THEN
	// if so, add our node first and jump out as done.
	nodesInExecutionOrder.AddFirst(Node);
	RETURN;
END_IF

// if not empty, then is our node higher priorty than the first in the list. 
nodesInExecutionOrder.First.TryGet(currentNode); 
IF currentNode.Order > Node.Order THEN
	// if yes, we are now first, jump out as done. 
	nodesInExecutionOrder.AddFirst(Node);
	RETURN;
END_IF

// here, the list has something in it, and we have less priority than the node in first place.

// get the last node in the list and remember this as "currentPosition" 
currentPosition := nodesInExecutionOrder.Last;

WHILE (TRUE) DO
	
	currentPosition.TryGet(currentNode); 
	// is the current position higer priority than our node?
	IF currentNode.Order <= Node.Order THEN
		// if so, then we go after, jump out as we are done. 
		nodesInExecutionOrder.AddAfter(currentPosition, Node);
		RETURN;
	END_IF
	
	// move one up the list towards the top and try again.
	currentPosition := currentPosition.Previous;

END_WHILE
END_METHOD

METHOD PUBLIC Accept
VAR_INPUT
	Visitor : I_NodeVisitor;
END_VAR
VAR
	enumerator : I_ForwardEnumerator;
	node : I_Node;
END_VAR
enumerator := nodes.GetEnumerator();

WHILE (enumerator.MoveNext()) DO
	
	IF enumerator.TryGet(node) THEN
		node.Accept(Visitor);
	END_IF

END_WHILE

enumerator.Dispose();
END_METHOD

METHOD PUBLIC AddNode
VAR_INPUT
	Node : I_Node;
END_VAR
nodes.AddOrUpdate(Node.id, Node);
UpdateExecutionOrder(Node);
EmitOnNodeAddedEvent(Node);
CreateExecuteEnumerator();
END_METHOD

METHOD PUBLIC Execute
VAR_INPUT
END_VAR
VAR
	node : I_Node;
END_VAR
executeEnumerator.Reset();

WHILE executeEnumerator.MoveNext() DO
	IF executeEnumerator.TryGet(node) THEN
		node.Execute();
	END_IF
END_WHILE
END_METHOD

METHOD PUBLIC GetNodesInOrderEnumerator : I_ForwardEnumerator
VAR_INPUT
END_VAR
GetNodesInOrderEnumerator := nodesInExecutionOrder.GetEnumerator();
END_METHOD

PROPERTY PUBLIC HasNodes : BOOL
GET
//HasNodes := NOT nodes.IsEmpty;
HasNodes := NOT nodes.IsEmpty OR NOT nodesInExecutionOrder.IsEmpty;
END_GET
END_PROPERTY

METHOD PUBLIC RemoveNode
VAR_INPUT
	Node : I_Node;
END_VAR
nodes.Remove(Node.Id);
nodesInExecutionOrder.Remove(Node);
CreateExecuteEnumerator();
END_METHOD

METHOD PUBLIC SerializeWith
VAR_INPUT
	Serializer : I_Serializer;
END_VAR
VAR
	enumerator : I_ForwardEnumerator;
	node : I_Node;
END_VAR
IF nodes.Count = 0 THEN
	RETURN;
END_IF

Serializer.AddKey('nodes');
Serializer.StartArray();

enumerator := nodes.GetEnumerator();

WHILE enumerator.MoveNext() DO
	IF enumerator.TryGet(node) THEN
		node.SerializeWith(Serializer);
	END_IF
END_WHILE

Serializer.EndArray();
enumerator.Dispose();
END_METHOD

METHOD PUBLIC TryDeserializeFrom : BOOL
VAR_INPUT
	Deserializer : I_Deserializer;
	Feedback : I_DeserializerFeedback;
END_VAR
VAR
	nodeDeserializer : I_Deserializer;
	nodesEnumerator : I_DeserializerArrayForwardEnumerator;
	nodeId : T_MAXSTRING;
	node : I_Node;
END_VAR
nodeDeserializer := Deserializer.GetKeyArray('nodes');
nodesEnumerator := nodeDeserializer.GetArrayEnumerator();

WHILE nodesEnumerator.MoveNext() DO
	
	IF NOT nodesEnumerator.Current.TryGetKeyString('id', nodeId, Feedback) THEN
		CONTINUE;
	END_IF
	
	IF NOT TryGetNodeById(nodeId, node)THEN
		CONTINUE;
	END_IF
	
	node.TryDeserializeFrom(nodesEnumerator.Current, Feedback);

END_WHILE

nodesEnumerator.Dispose();
END_METHOD

METHOD PUBLIC TryGetNodeById : BOOL
VAR_INPUT
	Id : T_MAXSTRING;
	Destination : REFERENCE TO I_Node;
END_VAR
VAR
	node : I_Node;
END_VAR
IF NOT nodes.TryGetValue(Id, node) THEN
	RETURN;
END_IF

Destination := node;
TryGetNodeById := TRUE;
END_METHOD

END_FUNCTION_BLOCK

// Node/Events/NodeAddedEvent
{attribute 'linkalways'} 
{attribute 'no_explicit_call' := 'This FB is a CLASS and must be accessed using methods or properties'}
{attribute 'enable_dynamic_creation'}
FUNCTION_BLOCK NodeAddedEvent EXTENDS Disposable IMPLEMENTS I_NodeAddedEvent
VAR
	_target : I_Node;
END_VAR

METHOD FB_init : BOOL
VAR_INPUT
	bInitRetains : BOOL; // if TRUE, the retain variables are initialized (warm start / cold start)
	bInCopyCode : BOOL;  // if TRUE, the instance afterwards gets moved into the copy code (online change)
	Target : I_Node;
END_VAR
THIS^._target := Target;
END_METHOD

PROPERTY PUBLIC Target : I_Node
GET
Target := _target;
END_GET
END_PROPERTY

END_FUNCTION_BLOCK

// Node/Events/I_NodeAddedEvent
INTERFACE I_NodeAddedEvent EXTENDS I_Event

PROPERTY PUBLIC Target : I_Node
GET
END_GET
END_PROPERTY

END_INTERFACE

// Link/Collection/NodeLinks
{attribute 'linkalways'} 
{attribute 'no_explicit_call' := 'This FB is a CLASS and must be accessed using methods or properties'}
{attribute 'enable_dynamic_creation'}
FUNCTION_BLOCK NodeLinks EXTENDS disposable IMPLEMENTS I_NodeLinks
VAR
	links : OrderedDictionary;
END_VAR

METHOD FB_exit : BOOL
VAR_INPUT
	bInCopyCode : BOOL; // if TRUE, the exit method is called for exiting an instance that is copied afterwards (online change).
END_VAR
IF bInCopyCode THEN
	RETURN;
END_IF

Clear();
END_METHOD

METHOD PRIVATE CreateNewLink : I_NodeLink
VAR_INPUT
	LinkId : T_MAXSTRING;
	LinkSourceNode : I_Node;
	LinkSource : I_LinkSource;
	LinkDestinationNode : I_Node;
	LinkDestination : I_LinkDestination;
END_VAR
VAR
	pLink : POINTER TO Link;
END_VAR
pLink := __NEW(
	Link(
		Id := LinkId, 
		SourceNode := LinkSourceNode,
		Source := LinkSource,
		DestinationNode := LinkDestinationNode,
		Destination := LinkDestination
	)
);

CreateNewLink := pLink^;
END_METHOD

METHOD PUBLIC Clear
VAR_INPUT
END_VAR
VAR
	enumerator : I_ForwardEnumerator;
	link : I_NodeLink;
END_VAR
enumerator := links.GetEnumerator();

WHILE (enumerator.MoveNext()) DO
	
	IF enumerator.TryGet(link) THEN
		link.Dispose();
	END_IF

END_WHILE

enumerator.Dispose();
links.Clear();
END_METHOD

METHOD PUBLIC Create : I_NodeLink
VAR_INPUT
	LinkId : T_MAXSTRING;
	LinkSourceNode : I_Node;
	LinkSource : I_LinkSource;
	LinkDestinationNode : I_Node;
	LinkDestination : I_LinkDestination;
END_VAR
VAR
	link : I_NodeLink;
END_VAR
link := CreateNewLink(
	LinkId, 
	LinkSourceNode,
	LinkSource,
	LinkDestinationNode,
	LinkDestination
);

links.AddOrUpdate(link.Id, link);
Create := link;
END_METHOD

METHOD PUBLIC DisconnectAll
VAR_INPUT
END_VAR
VAR
	enumerator : I_ForwardEnumerator;
	link : I_NodeLink;
END_VAR
enumerator := links.GetEnumerator();

WHILE (enumerator.MoveNext()) DO
	
	IF enumerator.TryGet(link) THEN
		link.Disconnect();
	END_IF

END_WHILE

enumerator.Dispose();
END_METHOD

METHOD PUBLIC GetKeyValueEnumerator : I_KeyValueForwardEnumerator
VAR_INPUT
END_VAR
GetKeyValueEnumerator := links.GetKeyValueEnumerator();
END_METHOD

METHOD PUBLIC TryGetLinkById : BOOL
VAR_INPUT
	Id : T_MAXSTRING;
	Destination : REFERENCE TO I_NodeLink;
END_VAR
VAR
	link : I_NodeLink;
END_VAR
IF NOT links.TryGetValue(Id, link) THEN
	RETURN;
END_IF

Destination := link;
TryGetLinkById := TRUE;
END_METHOD

END_FUNCTION_BLOCK

// Link/Interface/I_NodeLinks
INTERFACE I_NodeLinks EXTENDS I_Disposable

METHOD PUBLIC Clear
VAR_INPUT
END_VAR
END_METHOD

METHOD PUBLIC Create : I_NodeLink
VAR_INPUT
	LinkId : T_MAXSTRING;
	LinkSourceNode : I_Node;
	LinkSource : I_LinkSource;
	LinkDestinationNode : I_Node;
	LinkDestination : I_LinkDestination;
END_VAR
END_METHOD

METHOD PUBLIC DisconnectAll
VAR_INPUT
END_VAR
END_METHOD

METHOD PUBLIC GetKeyValueEnumerator : I_KeyValueForwardEnumerator
VAR_INPUT
END_VAR
END_METHOD

METHOD PUBLIC TryGetLinkById : BOOL
VAR_INPUT
	Id : T_MAXSTRING;
	Destination : REFERENCE TO I_NodeLink;
END_VAR
END_METHOD

END_INTERFACE

// Link/Interface/I_NodeLink
INTERFACE I_NodeLink EXTENDS I_Disposable

PROPERTY PUBLIC Destination : I_LinkDestination
GET
END_GET
END_PROPERTY

PROPERTY PUBLIC DestinationNode : I_Node
GET
END_GET
END_PROPERTY

METHOD PUBLIC Disconnect
VAR_INPUT
END_VAR
END_METHOD

PROPERTY PUBLIC Id : T_MAXSTRING
GET
END_GET
END_PROPERTY

PROPERTY PUBLIC Source : I_LinkSource
GET
END_GET
END_PROPERTY

PROPERTY PUBLIC SourceNode : I_Node
GET
END_GET
END_PROPERTY

METHOD PUBLIC TryConnect : BOOL;
VAR_INPUT
END_VAR
END_METHOD

END_INTERFACE

// Link/Link
{attribute 'linkalways'} 
{attribute 'no_explicit_call' := 'This FB is a CLASS and must be accessed using methods or properties'}
{attribute 'enable_dynamic_creation'}
FUNCTION_BLOCK Link EXTENDS Disposable IMPLEMENTS I_NodeLink
VAR
	_id : T_MAXSTRING;
	_sourceNode : I_Node;
	_source : I_LinkSource;
	_destinationNode : I_Node;
	_destination : I_LinkDestination;
END_VAR

METHOD FB_init : BOOL
VAR_INPUT
	bInitRetains : BOOL; // if TRUE, the retain variables are initialized (warm start / cold start)
	bInCopyCode : BOOL;  // if TRUE, the instance afterwards gets moved into the copy code (online change)
	Id : T_MAXSTRING;
	SourceNode : I_Node;
	Source : I_LinkSource;
	DestinationNode : I_Node;
	Destination : I_LinkDestination;
END_VAR
_id := Id;
_sourceNode := SourceNode;
_source := Source;
_destinationNode := DestinationNode;
_destination := Destination;
END_METHOD

METHOD FB_exit : BOOL
VAR_INPUT
	bInCopyCode : BOOL; // if TRUE, the exit method is called for exiting an instance that is copied afterwards (online change).
END_VAR
IF bInCopyCode THEN
	RETURN;
END_IF

Disconnect();
END_METHOD

PROPERTY PUBLIC Destination : I_LinkDestination
GET
Destination := _destination;
END_GET
END_PROPERTY

PROPERTY PUBLIC DestinationNode : I_Node
GET
DestinationNode := _destinationNode;
END_GET
END_PROPERTY

METHOD PUBLIC Disconnect
VAR_INPUT
END_VAR
IF _source = 0 THEN
	RETURN;
END_IF

IF _destination = 0 THEN
	RETURN;
END_IF

_destination.Disconnect();
END_METHOD

PROPERTY PUBLIC Id : T_MAXSTRING
GET
Id := _id;
END_GET
END_PROPERTY

PROPERTY PUBLIC Source : I_LinkSource
GET
Source := _source;
END_GET
END_PROPERTY

PROPERTY PUBLIC SourceNode : I_Node
GET
SourceNode := _sourceNode;
END_GET
END_PROPERTY

METHOD PUBLIC TryConnect : BOOL;
VAR_INPUT
END_VAR
IF _source = 0 THEN
	RETURN;
END_IF

IF _destination = 0 THEN
	RETURN;
END_IF

TryConnect := _destination.TryConnectTo(_source);
END_METHOD

END_FUNCTION_BLOCK

// Errors/MissingNodePrototypeDeserializationError
{attribute 'linkalways'} 
{attribute 'no_explicit_call' := 'This FB is a CLASS and must be accessed using methods or properties'}
{attribute 'enable_dynamic_creation'}
FUNCTION_BLOCK MissingNodePrototypeDeserializationError EXTENDS Error
VAR
	nodeType : T_MAXSTRING;
END_VAR

METHOD FB_init : BOOL
VAR_INPUT
	bInitRetains : BOOL; // if TRUE, the retain variables are initialized (warm start / cold start)
	bInCopyCode : BOOL;  // if TRUE, the instance afterwards gets moved into the copy code (online change)
	MissingType : T_MAXSTRING;
END_VAR
nodeType := MissingType;
END_METHOD

PROPERTY PUBLIC ErrorType : T_MAXSTRING
GET
ErrorType := 'MISSING_NODE_PROTOTYPE_DESERIALIZATION_ERROR';
END_GET
END_PROPERTY

PROPERTY PUBLIC Message : T_MAXSTRING
GET
Message := CONCAT('Deserialization Failed, Missing Node Prototype : ',nodeType);
END_GET
END_PROPERTY

END_FUNCTION_BLOCK

// Graph/Interfaces/I_Graphs
INTERFACE I_Graphs

METHOD PUBLIC Accept
VAR_INPUT
	visitor : I_GraphVisitor;
END_VAR
END_METHOD

METHOD PUBLIC AddGraph
VAR_INPUT
	Graph : I_Graph;
END_VAR
END_METHOD

METHOD PUBLIC DisposeAll
VAR_INPUT
END_VAR
END_METHOD

METHOD PUBLIC Execute
VAR_INPUT
END_VAR
END_METHOD

METHOD PUBLIC RemoveGraph
VAR_INPUT
	Graph : I_Graph;
END_VAR
END_METHOD

METHOD PUBLIC TryGetGraphByUuid : BOOL
VAR_INPUT
	Uuid : T_MAXSTRING;
	Destination : REFERENCE TO I_Graph;
END_VAR
END_METHOD

END_INTERFACE

// API/Visitors/GetStatusVisitor
{attribute 'linkalways'} 
{attribute 'no_explicit_call' := 'This FB is a CLASS and must be accessed using methods or properties'}
{attribute 'enable_dynamic_creation'}
FUNCTION_BLOCK GetStatusVisitor IMPLEMENTS I_GraphVisitor, I_NodeVisitor, I_ExtensionVisitor, I_ContentVisitor, I_AlarmVisitor
VAR
	serializer : I_Serializer;
END_VAR

METHOD PUBLIC Initialize
VAR_INPUT
	Serializer : I_Serializer;
END_VAR
THIS^.serializer := Serializer;
END_METHOD

METHOD VisitAlarm
VAR_INPUT
	VisitingAlarm : I_Alarm;
END_VAR
IF VisitingAlarm.Active THEN
	serializer.StartObject();
	serializer.AddKeyString('message', VisitingAlarm.Message);
	serializer.AddKeyString('reason', VisitingAlarm.Reason);
	serializer.EndObject();
END_IF
END_METHOD

METHOD VisitContent
VAR_INPUT
	VisitingContent : I_Content;
END_VAR
serializer.StartObject();

serializer.AddKeyString('name', VisitingContent.Name);
serializer.AddKeyObject('value', VisitingContent.Data);

serializer.EndObject();
END_METHOD

METHOD VisitExtension
VAR_INPUT
	VisitingExtension : I_Extension;
END_VAR
Serializer.StartObject();
Serializer.AddKeyString('name', VisitingExtension.Name);

IF VisitingExtension.Alarms.HasAlarms THEN
	serializer.addkey('alarms');
	serializer.StartArray();
	VisitingExtension.Alarms.Accept(THIS^);
	serializer.EndArray();
END_IF

IF VisitingExtension.Contents.HasContents THEN
	serializer.addkey('contents');
	serializer.StartArray();
	VisitingExtension.Contents.Accept(THIS^);
	serializer.EndArray();
END_IF

Serializer.EndObject();
END_METHOD

METHOD VisitGraph
VAR_INPUT
	VisitingGraph : I_Graph;
END_VAR
VAR
	includeInGetStatusVisitor : IncludeInGetStatusVisitor;
END_VAR
serializer.StartObject();

serializer.addKeyString('uuid', VisitingGraph.Uuid);

IF VisitingGraph.Alarms.HasRaisedAlarm THEN
	serializer.addkey('alarms');
	serializer.StartArray();
	VisitingGraph.Alarms.Accept(THIS^);
	serializer.EndArray();
END_IF

IF includeInGetStatusVisitor.CheckExtensions(VisitingGraph) THEN
	serializer.addkey('extensions');
	serializer.StartArray();
	VisitingGraph.Extensions.Accept(THIS^);
	serializer.EndArray();
END_IF

IF VisitingGraph.Contents.HasContents THEN
	serializer.addkey('contents');
	serializer.StartArray();
	VisitingGraph.Contents.Accept(THIS^);
	serializer.EndArray();
END_IF

IF VisitingGraph.Nodes.HasNodes THEN
	serializer.addkey('nodes');
	serializer.StartArray();
	VisitingGraph.Nodes.Accept(THIS^);
	serializer.EndArray();
END_IF

serializer.EndObject();
END_METHOD

METHOD VisitNode
VAR_INPUT
	VisitingNode : I_Node;
END_VAR
VAR
	includeInGetStatusVisitor : IncludeInGetStatusVisitor;
END_VAR
IF NOT includeInGetStatusVisitor.CheckNode(VisitingNode) THEN
	RETURN;
END_IF

serializer.StartObject();
serializer.addKeyString('id', VisitingNode.Id);

IF VisitingNode.Alarms.HasRaisedAlarm THEN
	serializer.addkey('alarms');
	serializer.StartArray();
	VisitingNode.Alarms.Accept(THIS^);
	serializer.EndArray();
END_IF

IF includeInGetStatusVisitor.CheckExtensions(VisitingNode) THEN
	serializer.addkey('extensions');
	serializer.StartArray();
	VisitingNode.Extensions.Accept(THIS^);
	serializer.EndArray();
END_IF

IF VisitingNode.Contents.HasContents THEN
	serializer.addkey('contents');
	serializer.StartArray();
	VisitingNode.Contents.Accept(THIS^);
	serializer.EndArray();
END_IF

serializer.EndObject();
END_METHOD

END_FUNCTION_BLOCK

// API/Visitors/IncludeInGetStatusVisitor
{attribute 'linkalways'} 
{attribute 'no_explicit_call' := 'This FB is a CLASS and must be accessed using methods or properties'}
{attribute 'enable_dynamic_creation'}
FUNCTION_BLOCK IncludeInGetStatusVisitor IMPLEMENTS I_NodeVisitor, I_ExtensionVisitor
VAR
	shouldInclude : BOOL;
END_VAR

METHOD PUBLIC CheckExtensions : BOOL;
VAR_INPUT
	ExtensionHost : I_HostExtensions;
END_VAR
shouldInclude := FALSE;
ExtensionHost.Extensions.Accept(THIS^);
CheckExtensions := shouldInclude;
END_METHOD

METHOD PUBLIC CheckNode : BOOL;
VAR_INPUT
	Node : I_Node;
END_VAR
shouldInclude := FALSE;
Node.Accept(THIS^);
CheckNode := shouldInclude;
END_METHOD

METHOD VisitExtension
VAR_INPUT
	VisitingExtension : I_Extension;
END_VAR
IF VisitingExtension.Contents.HasContents THEN
	shouldInclude := TRUE;
	RETURN;
END_IF

IF VisitingExtension.Alarms.HasRaisedAlarm THEN
	shouldInclude := TRUE;
	RETURN;
END_IF
END_METHOD

METHOD VisitNode
VAR_INPUT
	VisitingNode : I_Node;
END_VAR
IF VisitingNode.Contents.HasContents THEN
	shouldInclude := TRUE;
	RETURN;
END_IF

IF VisitingNode.Alarms.HasRaisedAlarm THEN
	shouldInclude := TRUE;
	RETURN;
END_IF

IF VisitingNode.Extensions.HasExtensions THEN
	VisitingNode.Extensions.Accept(THIS^);
END_IF
END_METHOD

END_FUNCTION_BLOCK

// API/Handlers/GetBlueprintsRpcHandler
{attribute 'linkalways'} 
{attribute 'no_explicit_call' := 'This FB is a CLASS and must be accessed using methods or properties'}
{attribute 'enable_dynamic_creation'}
FUNCTION_BLOCK GetBlueprintsRpcHandler IMPLEMENTS I_AsynchronousRpcHandler
VAR
	nodeFactory : I_NodeFactory;
END_VAR

METHOD Handle
VAR_INPUT
	Parameters : I_Deserializer;
	Response : I_AsynchronousRpcResponse;
END_VAR
VAR
	getBlueprintsVisitor : GetBlueprintsVisitor;
	getPaginatedBlueprintsVisitor : GetPaginatedBlueprintsVisitor;
	visitor : I_NodeFactoryVisitor;
	serializer : I_Serializer;
	feedback : DeserializerFeedback;
	offset : UDINT;
	maxLimit : UDINT;
END_VAR
IF nodeFactory = 0 THEN
	Response.RejectWithMessage('GetBlueprintsRpcHandler has not been initialized with a valid nodeFactory object');
	RETURN;
END_IF

serializer := Response.GetSerializer();

IF Parameters.TryGetKeyUdint('offset', offset, feedback) AND_THEN Parameters.TryGetKeyUdint('limit', maxLimit, feedback) THEN
	// if the offset and limit are provide then use the paginated visitor
	getPaginatedBlueprintsVisitor.Initialize(serializer, offset, maxlimit);
	visitor := getPaginatedBlueprintsVisitor;
ELSE
	// if the offset and limit are not supplied then try to get all blueprints
	getBlueprintsVisitor.Initialize(serializer);
	visitor := getBlueprintsVisitor;
END_IF

nodeFactory.Accept(visitor);
Response.CompleteWithSerializer(serializer);
serializer.Dispose();
END_METHOD

METHOD PUBLIC Initialize
VAR_INPUT
	NodeFactory : I_NodeFactory;
END_VAR
THIS^.nodeFactory := NodeFactory;
END_METHOD

END_FUNCTION_BLOCK

// API/Visitors/GetPaginatedBlueprintsVisitor
{attribute 'linkalways'} 
{attribute 'no_explicit_call' := 'This FB is a CLASS and must be accessed using methods or properties'}
{attribute 'enable_dynamic_creation'}
FUNCTION_BLOCK GetPaginatedBlueprintsVisitor IMPLEMENTS I_NodeFactoryVisitor, I_NodePrototypeVisitor, I_NodeVisitor, I_ExtensionVisitor, I_InputPortVisitor, I_OutputPortVisitor, I_MetadataVisitor, I_ContentVisitor, I_ParameterVisitor, I_AlarmVisitor
VAR
	serializer : I_Serializer;
	offset : UDINT;
	maxLimit : UDINT;
	
	// used to track count
	currentIndex : UDINT;
	endIndex : UDINT;
	blueprintsCollected : UDINT;
	totalBlueprints : UDINT;
END_VAR

METHOD PUBLIC Initialize
VAR_INPUT
	Serializer : I_Serializer;
	Offset : UDINT;
	MaxLimit : UDINT;
END_VAR
THIS^.serializer := Serializer;
THIS^.offset := Offset;
THIS^.maxLimit := MaxLimit;

THIS^.currentIndex := 0;
THIS^.endIndex := Offset + MaxLimit -1;

THIS^.blueprintsCollected := 0;
THIS^.totalBlueprints := 0;
END_METHOD

METHOD VisitAlarm
VAR_INPUT
	VisitingAlarm : I_Alarm;
END_VAR
serializer.AddString(VisitingAlarm.Message);
END_METHOD

METHOD VisitContent
VAR_INPUT
	VisitingContent : I_Content;
END_VAR
serializer.StartObject();

serializer.AddKeyString('name', VisitingContent.Name);
serializer.Addkey('datatype');
VisitingContent.Data.SerializeTypeWith(serializer);

IF VisitingContent.Metadatum.HasMetadata THEN
	serializer.addkey('metadata');
	serializer.StartArray();
	VisitingContent.Metadatum.Accept(THIS^);
	serializer.EndArray();
END_IF

serializer.EndObject();
END_METHOD

METHOD VisitExtension
VAR_INPUT
	VisitingExtension : I_Extension;
END_VAR
Serializer.StartObject();
Serializer.AddKeyString('name', VisitingExtension.Name);

IF VisitingExtension.Metadatum.HasMetadata THEN
	serializer.addkey('metadata');
	serializer.StartArray();
	VisitingExtension.Metadatum.Accept(THIS^);
	serializer.EndArray();
END_IF

IF VisitingExtension.Alarms.HasAlarms THEN
	serializer.addkey('alarms');
	serializer.StartArray();
	VisitingExtension.Alarms.Accept(THIS^);
	serializer.EndArray();
END_IF

IF VisitingExtension.InputPorts.HasInputPorts THEN
	serializer.addkey('inputPorts');
	serializer.StartArray();
	VisitingExtension.InputPorts.Accept(THIS^);
	serializer.EndArray();
END_IF

IF VisitingExtension.OutputPorts.HasOutputPorts THEN
	serializer.addkey('outputPorts');
	serializer.StartArray();
	VisitingExtension.OutputPorts.Accept(THIS^);
	serializer.EndArray();
END_IF

IF VisitingExtension.Parameters.HasParameters THEN
	serializer.addkey('parameters');
	serializer.StartArray();
	VisitingExtension.Parameters.Accept(THIS^);
	serializer.EndArray();
END_IF

IF VisitingExtension.Contents.HasContents THEN
	serializer.addkey('contents');
	serializer.StartArray();
	VisitingExtension.Contents.Accept(THIS^);
	serializer.EndArray();
END_IF

Serializer.EndObject();
END_METHOD

METHOD VisitInputPort
VAR_INPUT
	VisitingInputPort : I_InputPort;
END_VAR
serializer.StartObject();

serializer.AddKeyString('name', VisitingInputPort.Name);
serializer.Addkey('datatype');
VisitingInputPort.Data.SerializeTypeWith(serializer);

IF VisitingInputPort.Metadatum.HasMetadata THEN
	serializer.addkey('metadata');
	serializer.StartArray();
	VisitingInputPort.Metadatum.Accept(THIS^);
	serializer.EndArray();
END_IF

serializer.EndObject();
END_METHOD

METHOD VisitMetadatum
VAR_INPUT
	VisitingMetadatum : I_Metadata;
END_VAR
serializer.StartObject();
serializer.AddKeyString('name', VisitingMetadatum.Name);
serializer.AddkeyObject('value', VisitingMetadatum.Data);
serializer.EndObject();
END_METHOD

METHOD VisitNode
VAR_INPUT
	VisitingNode : I_Node;
END_VAR
serializer.StartObject();

IF VisitingNode.Metadatum.HasMetadata THEN
	serializer.addkey('metadata');
	serializer.StartArray();
	VisitingNode.Metadatum.Accept(THIS^);
	serializer.EndArray();
END_IF

IF VisitingNode.Alarms.HasAlarms THEN
	serializer.addkey('alarms');
	serializer.StartArray();
	VisitingNode.Alarms.Accept(THIS^);
	serializer.EndArray();
END_IF

IF VisitingNode.Extensions.HasExtensions THEN
	serializer.addkey('extensions');
	serializer.StartArray();
	VisitingNode.Extensions.Accept(THIS^);
	serializer.EndArray();
END_IF

IF VisitingNode.InputPorts.HasInputPorts THEN
	serializer.addkey('inputPorts');
	serializer.StartArray();
	VisitingNode.InputPorts.Accept(THIS^);
	serializer.EndArray();
END_IF

IF VisitingNode.OutputPorts.HasOutputPorts THEN
	serializer.addkey('outputPorts');
	serializer.StartArray();
	VisitingNode.OutputPorts.Accept(THIS^);
	serializer.EndArray();
END_IF

IF VisitingNode.Parameters.HasParameters THEN
	serializer.addkey('parameters');
	serializer.StartArray();
	VisitingNode.Parameters.Accept(THIS^);
	serializer.EndArray();
END_IF

IF VisitingNode.Contents.HasContents THEN
	serializer.addkey('contents');
	serializer.StartArray();
	VisitingNode.Contents.Accept(THIS^);
	serializer.EndArray();
END_IF

serializer.EndObject();
END_METHOD

METHOD VisitNodeFactory
VAR_INPUT
	VisitingNodeFactory : I_NodeFactory;
END_VAR
serializer.StartObject();
serializer.AddKey('blueprints');
serializer.StartArray();
VisitingNodeFactory.NodePrototypes.Accept(THIS^);
serializer.EndArray();
serializer.AddKeyUdint('returnedCount', blueprintsCollected);
serializer.AddKeyUdint('totalCount', totalBlueprints);
serializer.AddKeyUdint('nextOffset', offset + blueprintsCollected);
serializer.AddKeyBool('hasMore', offset + blueprintsCollected < totalBlueprints); 
serializer.EndObject();
END_METHOD

METHOD VisitNodePrototype
VAR_INPUT
	VisitingPrototype : I_NodePrototype;
END_VAR
// we're not yet in range of collection
IF currentIndex < offset THEN
	currentIndex := currentIndex + 1;
	totalBlueprints := totalBlueprints + 1;
	RETURN;
END_IF

// we're over range of the collection
IF currentIndex > endIndex THEN
	currentIndex := currentIndex + 1;
	totalBlueprints := totalBlueprints + 1;
	RETURN;
END_IF

// we're in the range to collect. 

blueprintsCollected := blueprintsCollected + 1;
currentIndex := currentIndex + 1;
totalBlueprints := totalBlueprints + 1;

serializer.StartObject();
serializer.AddKeyString('path', VisitingPrototype.Path);
serializer.AddKey('node');
VisitingPrototype.Node.Accept(THIS^);
serializer.EndObject();
END_METHOD

METHOD VisitOutputPort
VAR_INPUT
	VisitingOutputPort : I_OutputPort;
END_VAR
serializer.StartObject();

serializer.AddKeyString('name', VisitingOutputPort.Name);
serializer.Addkey('datatype');
VisitingOutputPort.Data.SerializeTypeWith(serializer);

IF VisitingOutputPort.Metadatum.HasMetadata THEN
	serializer.addkey('metadata');
	serializer.StartArray();
	VisitingOutputPort.Metadatum.Accept(THIS^);
	serializer.EndArray();
END_IF

serializer.EndObject();
END_METHOD

METHOD VisitParameter
VAR_INPUT
	VisitingProperty : I_Parameter;
END_VAR
serializer.StartObject();

serializer.AddKeyString('name', VisitingProperty.Name);
serializer.Addkey('datatype');
VisitingProperty.Data.SerializeTypeWith(serializer);
serializer.Addkey('defaultValue');
VisitingProperty.Data.SerializeWith(serializer);

IF VisitingProperty.Metadatum.HasMetadata THEN
	serializer.addkey('metadata');
	serializer.StartArray();
	VisitingProperty.Metadatum.Accept(THIS^);
	serializer.EndArray();
END_IF

Serializer.EndObject();
END_METHOD

END_FUNCTION_BLOCK

// API/Visitors/GetBlueprintsVisitor
{attribute 'linkalways'} 
{attribute 'no_explicit_call' := 'This FB is a CLASS and must be accessed using methods or properties'}
{attribute 'enable_dynamic_creation'}
FUNCTION_BLOCK GetBlueprintsVisitor IMPLEMENTS I_NodeFactoryVisitor, I_NodePrototypeVisitor, I_NodeVisitor, I_ExtensionVisitor, I_InputPortVisitor, I_OutputPortVisitor, I_MetadataVisitor, I_ContentVisitor, I_ParameterVisitor, I_AlarmVisitor
VAR
	serializer : I_Serializer;
END_VAR

METHOD PUBLIC Initialize
VAR_INPUT
	Serializer : I_Serializer;
END_VAR
THIS^.serializer := Serializer;
END_METHOD

METHOD VisitAlarm
VAR_INPUT
	VisitingAlarm : I_Alarm;
END_VAR
serializer.AddString(VisitingAlarm.Message);
END_METHOD

METHOD VisitContent
VAR_INPUT
	VisitingContent : I_Content;
END_VAR
serializer.StartObject();

serializer.AddKeyString('name', VisitingContent.Name);
serializer.Addkey('datatype');
VisitingContent.Data.SerializeTypeWith(serializer);

IF VisitingContent.Metadatum.HasMetadata THEN
	serializer.addkey('metadata');
	serializer.StartArray();
	VisitingContent.Metadatum.Accept(THIS^);
	serializer.EndArray();
END_IF

serializer.EndObject();
END_METHOD

METHOD VisitExtension
VAR_INPUT
	VisitingExtension : I_Extension;
END_VAR
Serializer.StartObject();
Serializer.AddKeyString('name', VisitingExtension.Name);

IF VisitingExtension.Metadatum.HasMetadata THEN
	serializer.addkey('metadata');
	serializer.StartArray();
	VisitingExtension.Metadatum.Accept(THIS^);
	serializer.EndArray();
END_IF

IF VisitingExtension.Alarms.HasAlarms THEN
	serializer.addkey('alarms');
	serializer.StartArray();
	VisitingExtension.Alarms.Accept(THIS^);
	serializer.EndArray();
END_IF

IF VisitingExtension.InputPorts.HasInputPorts THEN
	serializer.addkey('inputPorts');
	serializer.StartArray();
	VisitingExtension.InputPorts.Accept(THIS^);
	serializer.EndArray();
END_IF

IF VisitingExtension.OutputPorts.HasOutputPorts THEN
	serializer.addkey('outputPorts');
	serializer.StartArray();
	VisitingExtension.OutputPorts.Accept(THIS^);
	serializer.EndArray();
END_IF

IF VisitingExtension.Parameters.HasParameters THEN
	serializer.addkey('parameters');
	serializer.StartArray();
	VisitingExtension.Parameters.Accept(THIS^);
	serializer.EndArray();
END_IF

IF VisitingExtension.Contents.HasContents THEN
	serializer.addkey('contents');
	serializer.StartArray();
	VisitingExtension.Contents.Accept(THIS^);
	serializer.EndArray();
END_IF

Serializer.EndObject();
END_METHOD

METHOD VisitInputPort
VAR_INPUT
	VisitingInputPort : I_InputPort;
END_VAR
serializer.StartObject();

serializer.AddKeyString('name', VisitingInputPort.Name);
serializer.Addkey('datatype');
VisitingInputPort.Data.SerializeTypeWith(serializer);

IF VisitingInputPort.Metadatum.HasMetadata THEN
	serializer.addkey('metadata');
	serializer.StartArray();
	VisitingInputPort.Metadatum.Accept(THIS^);
	serializer.EndArray();
END_IF

serializer.EndObject();
END_METHOD

METHOD VisitMetadatum
VAR_INPUT
	VisitingMetadatum : I_Metadata;
END_VAR
serializer.StartObject();
serializer.AddKeyString('name', VisitingMetadatum.Name);
serializer.AddkeyObject('value', VisitingMetadatum.Data);
serializer.EndObject();
END_METHOD

METHOD VisitNode
VAR_INPUT
	VisitingNode : I_Node;
END_VAR
serializer.StartObject();

IF VisitingNode.Metadatum.HasMetadata THEN
	serializer.addkey('metadata');
	serializer.StartArray();
	VisitingNode.Metadatum.Accept(THIS^);
	serializer.EndArray();
END_IF

IF VisitingNode.Alarms.HasAlarms THEN
	serializer.addkey('alarms');
	serializer.StartArray();
	VisitingNode.Alarms.Accept(THIS^);
	serializer.EndArray();
END_IF

IF VisitingNode.Extensions.HasExtensions THEN
	serializer.addkey('extensions');
	serializer.StartArray();
	VisitingNode.Extensions.Accept(THIS^);
	serializer.EndArray();
END_IF

IF VisitingNode.InputPorts.HasInputPorts THEN
	serializer.addkey('inputPorts');
	serializer.StartArray();
	VisitingNode.InputPorts.Accept(THIS^);
	serializer.EndArray();
END_IF

IF VisitingNode.OutputPorts.HasOutputPorts THEN
	serializer.addkey('outputPorts');
	serializer.StartArray();
	VisitingNode.OutputPorts.Accept(THIS^);
	serializer.EndArray();
END_IF

IF VisitingNode.Parameters.HasParameters THEN
	serializer.addkey('parameters');
	serializer.StartArray();
	VisitingNode.Parameters.Accept(THIS^);
	serializer.EndArray();
END_IF

IF VisitingNode.Contents.HasContents THEN
	serializer.addkey('contents');
	serializer.StartArray();
	VisitingNode.Contents.Accept(THIS^);
	serializer.EndArray();
END_IF

serializer.EndObject();
END_METHOD

METHOD VisitNodeFactory
VAR_INPUT
	VisitingNodeFactory : I_NodeFactory;
END_VAR
serializer.StartObject();
serializer.AddKey('blueprints');
serializer.StartArray();
VisitingNodeFactory.NodePrototypes.Accept(THIS^);
serializer.EndArray();
serializer.EndObject();
END_METHOD

METHOD VisitNodePrototype
VAR_INPUT
	VisitingPrototype : I_NodePrototype;
END_VAR
serializer.StartObject();
serializer.AddKeyString('path', VisitingPrototype.Path);
serializer.AddKey('node');
VisitingPrototype.Node.Accept(THIS^);
serializer.EndObject();
END_METHOD

METHOD VisitOutputPort
VAR_INPUT
	VisitingOutputPort : I_OutputPort;
END_VAR
serializer.StartObject();

serializer.AddKeyString('name', VisitingOutputPort.Name);
serializer.Addkey('datatype');
VisitingOutputPort.Data.SerializeTypeWith(serializer);

IF VisitingOutputPort.Metadatum.HasMetadata THEN
	serializer.addkey('metadata');
	serializer.StartArray();
	VisitingOutputPort.Metadatum.Accept(THIS^);
	serializer.EndArray();
END_IF

serializer.EndObject();
END_METHOD

METHOD VisitParameter
VAR_INPUT
	VisitingProperty : I_Parameter;
END_VAR
serializer.StartObject();

serializer.AddKeyString('name', VisitingProperty.Name);
serializer.Addkey('datatype');
VisitingProperty.Data.SerializeTypeWith(serializer);
serializer.Addkey('defaultValue');
VisitingProperty.Data.SerializeWith(serializer);

IF VisitingProperty.Metadatum.HasMetadata THEN
	serializer.addkey('metadata');
	serializer.StartArray();
	VisitingProperty.Metadatum.Accept(THIS^);
	serializer.EndArray();
END_IF

Serializer.EndObject();
END_METHOD

END_FUNCTION_BLOCK

// API/Handlers/GetContentValueHandler
{attribute 'linkalways'} 
{attribute 'no_explicit_call' := 'This FB is a CLASS and must be accessed using methods or properties'}
{attribute 'enable_dynamic_creation'}
FUNCTION_BLOCK GetContentValueHandler IMPLEMENTS I_AsynchronousRpcHandler
VAR
	graphs : I_Graphs;
END_VAR

METHOD Handle
VAR_INPUT
	Parameters : I_Deserializer;
	Response : I_AsynchronousRpcResponse;
END_VAR
VAR
	graphUuid : T_MAXSTRING;
	nodeId : T_MAXSTRING;
	contentName : T_MAXSTRING;
	visitor : RetrieveNodeContentValue;
	serializer : I_Serializer;
	feedback : DeserializerFeedback;
END_VAR
IF NOT Parameters.TryGetKeyString('graphUuid', graphUuid, feedback) THEN
	Response.RejectWithMessage(feedback.FirstError.Message);
	RETURN;
END_IF

IF NOT Parameters.TryGetKeyString('nodeId', nodeId, feedback) THEN
	Response.RejectWithMessage(feedback.FirstError.Message);
	RETURN;
END_IF

IF NOT Parameters.TryGetKeyString('contentName', contentName, feedback) THEN
	Response.RejectWithMessage(feedback.FirstError.Message);
	RETURN;
END_IF

serializer := Response.GetSerializer();
visitor.Initialize(graphUuid, nodeId, contentName, serializer);
graphs.Accept(visitor);

IF visitor.Error THEN
	Response.RejectWithMessage(visitor.ErrorMessage);
	serializer.Dispose();
	RETURN;
END_IF

IF NOT visitor.Done THEN
	Response.RejectWithMessage('Invalid graphUuid');
	serializer.Dispose();
	RETURN;
END_IF

Response.CompleteWithSerializer(serializer);
serializer.Dispose();
END_METHOD

METHOD PUBLIC Initialize
VAR_INPUT
	Graphs : I_Graphs;
END_VAR
THIS^.graphs := Graphs;
END_METHOD

END_FUNCTION_BLOCK

// API/Visitors/RetrieveNodeContentValue
{attribute 'linkalways'} 
{attribute 'no_explicit_call' := 'This FB is a CLASS and must be accessed using methods or properties'}
{attribute 'enable_dynamic_creation'}
FUNCTION_BLOCK RetrieveNodeContentValue IMPLEMENTS I_GraphVisitor, I_NodeVisitor, I_ContentVisitor
VAR
	graphUuid : T_MAXSTRING;
	nodeId : T_MAXSTRING;
	contentName : T_MAXSTRING;
	serializer : I_Serializer;
	_done : BOOL;
	_error : BOOL;
	_errorMessage : T_MAXSTRING;
END_VAR

METHOD PRIVATE LogInvalidContentNameError
VAR_INPUT
END_VAR
_errorMessage := 'Invalid Content Name';
_error := TRUE;
END_METHOD

METHOD PRIVATE LogInvalidNodeIdError
VAR_INPUT
END_VAR
_errorMessage := 'Invalid Node Id';
_error := TRUE;
END_METHOD

METHOD PRIVATE Reset
VAR_INPUT
END_VAR
_done := FALSE;
_errorMessage := '';
_error := FALSE;
END_METHOD

PROPERTY PUBLIC Done : BOOL
GET
Done := _done;
END_GET
END_PROPERTY

PROPERTY PUBLIC Error : BOOL
GET
Error := _error;
END_GET
END_PROPERTY

PROPERTY PUBLIC ErrorMessage : T_MAXSTRING
GET
ErrorMessage := _errorMessage;
END_GET
END_PROPERTY

METHOD PUBLIC Initialize
VAR_INPUT
	GraphUuid : T_MAXSTRING;
	NodeId : T_MAXSTRING;
	ContentName : T_MAXSTRING;
	Serializer : I_Serializer;
END_VAR
THIS^.graphUuid := GraphUuid;
THIS^.nodeId := NodeId;
THIS^.contentName := ContentName;
THIS^.serializer := Serializer;
END_METHOD

METHOD VisitContent
VAR_INPUT
	VisitingContent : I_Content;
END_VAR
VisitingContent.SerializeWith(serializer);
END_METHOD

METHOD VisitGraph
VAR_INPUT
	VisitingGraph : I_Graph;
END_VAR
VAR
	node : I_Node;
END_VAR
Reset();

IF NOT (VisitingGraph.Uuid = graphUuid) THEN
	RETURN;
END_IF

IF NOT VisitingGraph.Nodes.TryGetNodeById(nodeId, node) THEN
	LogInvalidNodeIdError();
	RETURN;
END_IF

node.Accept(THIS^);
END_METHOD

METHOD VisitNode
VAR_INPUT
	VisitingNode : I_Node;
END_VAR
VAR
	content : I_Content;
END_VAR
IF NOT VisitingNode.Contents.TryGetContentByName(contentName, content) THEN
	LogInvalidContentNameError();
	RETURN;
END_IF

content.Accept(THIS^);
END_METHOD

END_FUNCTION_BLOCK

// API/Handlers/GetStatusRpcHandler
{attribute 'linkalways'} 
{attribute 'no_explicit_call' := 'This FB is a CLASS and must be accessed using methods or properties'}
{attribute 'enable_dynamic_creation'}
FUNCTION_BLOCK GetStatusRpcHandler IMPLEMENTS I_AsynchronousRpcHandler
VAR
	graphs : I_Graphs;
END_VAR

METHOD Handle
VAR_INPUT
	Parameters : I_Deserializer;
	Response : I_AsynchronousRpcResponse;
END_VAR
VAR
	graphUuid : T_MAXSTRING;
	graph : I_Graph;
	feedback : DeserializerFeedback;
	serializer : I_Serializer;
	getStatusVisitor : GetStatusVisitor;
END_VAR
IF NOT Parameters.TryGetKeyString('graphUuid', graphUuid, feedback) THEN
	Response.RejectWithMessage(feedback.FirstError.Message);
	RETURN;
END_IF

IF NOT graphs.TryGetGraphByUuid(graphUuid,graph) THEN
	Response.RejectWithMessage(concat('Unknown UUID : ', graphUuid));
	RETURN;
END_IF

serializer := Response.GetSerializer();
getStatusVisitor.Initialize(serializer);
getStatusVisitor.VisitGraph(graph);
Response.CompleteWithSerializer(serializer);
serializer.Dispose();
END_METHOD

METHOD PUBLIC Initialize
VAR_INPUT
	Graphs : I_Graphs;
END_VAR
THIS^.graphs := Graphs;
END_METHOD

END_FUNCTION_BLOCK

// API/Handlers/UpdateParameterValueHandler
{attribute 'linkalways'} 
{attribute 'no_explicit_call' := 'This FB is a CLASS and must be accessed using methods or properties'}
{attribute 'enable_dynamic_creation'}
FUNCTION_BLOCK UpdateParameterValueHandler IMPLEMENTS I_AsynchronousRpcHandler
VAR
	graphs : I_Graphs;
END_VAR

METHOD Handle
VAR_INPUT
	Parameters : I_Deserializer;
	Response : I_AsynchronousRpcResponse;
END_VAR
VAR
	graphUuid : T_MAXSTRING;
	graph : I_Graph;
	nodeId : T_MAXSTRING;
	node : I_Node;
	parameterName : T_MAXSTRING;
	parameter : I_Parameter;
	visitor : RetrieveNodeContentValue;
	serializer : I_Serializer;
	feedback : DeserializerFeedback;
END_VAR
IF NOT Parameters.TryGetKeyString('graphUuid', graphUuid, feedback) THEN
	Response.RejectWithMessage(feedback.FirstError.Message);
	RETURN;
END_IF

IF NOT graphs.TryGetGraphByUuid(graphUuid, graph) THEN
	Response.RejectWithMessage('Invalid or missing graphUuid');
	RETURN;
END_IF

IF NOT Parameters.TryGetKeyString('nodeId', nodeId, feedback) THEN
	Response.RejectWithMessage(feedback.FirstError.Message);
	RETURN;
END_IF

IF NOT graph.Nodes.TryGetNodeById(nodeId, node) THEN
	Response.RejectWithMessage('Invalid or missing nodeId');
	RETURN;
END_IF

IF NOT Parameters.TryGetKeyString('parameterName', parameterName, feedback) THEN
	Response.RejectWithMessage(feedback.FirstError.Message);
	RETURN;
END_IF

IF NOT node.Parameters.TryGetParameterByName(parameterName, parameter) THEN
	Response.RejectWithMessage('Invalid or missing parameterName');
	RETURN;
END_IF

IF NOT Parameters.TryDeserializeKeyToObject ('parameterValue', parameter, feedback) THEN
	Response.RejectWithMessage(feedback.FirstError.Message);
	RETURN;
END_IF

Response.CompleteWithString(graphUuid);
END_METHOD

METHOD PUBLIC Initialize
VAR_INPUT
	Graphs : I_Graphs;
END_VAR
THIS^.graphs := Graphs;
END_METHOD

END_FUNCTION_BLOCK

// API/GraphFrameworkApi
{attribute 'linkalways'} 
{attribute 'no_explicit_call' := 'This FB is a CLASS and must be accessed using methods or properties'}
{attribute 'enable_dynamic_creation'}
FUNCTION_BLOCK GraphFrameworkApi IMPLEMENTS I_RpcApi, I_HostGraphs, I_EventEmitter
VAR
	graphFramework : I_GraphFramework;
	eventEmitter : EventEmitter;
	graphHost : GraphHost(THIS^, eventEmitter);
	createGraphRpcHandler : CreateGraphRpcHandler;
	getStatusRpcHandler : GetStatusRpcHandler;
	getBlueprintsRpcHandler : GetBlueprintsRpcHandler;
	getContentValueHandler : GetContentValueHandler;
	updateParameterValueHandler : UpdateParameterValueHandler;
END_VAR

METHOD FB_init : BOOL
VAR_INPUT
	bInitRetains : BOOL; // if TRUE, the retain variables are initialized (warm start / cold start)
	bInCopyCode : BOOL;  // if TRUE, the instance afterwards gets moved into the copy code (online change)
	GraphFramework : I_GraphFramework;
END_VAR
THIS^.graphFramework := GraphFramework;

getBlueprintsRpcHandler.Initialize(GraphFramework.NodeFactory);
getStatusRpcHandler.Initialize(graphHost);
createGraphRpcHandler.Initialize(GraphFramework, graphHost);
getContentValueHandler.Initialize(graphHost);
updateParameterValueHandler.Initialize(graphHost);
END_METHOD

METHOD FB_exit : BOOL
VAR_INPUT
	bInCopyCode : BOOL; // if TRUE, the exit method is called for exiting an instance that is copied afterwards (online change).
END_VAR
IF bInCopyCode THEN
	RETURN;
END_IF

graphs.DisposeAll();
END_METHOD

METHOD PUBLIC CyclicCall
VAR_INPUT
END_VAR
graphHost.Execute();
END_METHOD

PROPERTY PUBLIC Graphs : I_Graphs
GET
Graphs := graphHost;
END_GET
END_PROPERTY

METHOD PUBLIC OffEvent
VAR_INPUT
	EventName : T_MaxString;
	EventHandler : I_EventHandler;
END_VAR
eventEmitter.OffEvent(EventName, EventHandler);
END_METHOD

